	VAR jointtarget CDP_2918 := [[-11.73, 36.5, 4.79, 0, 48.7, -293.98], [9E9, 9E9, 9E9, 9E9, 9E9, 9E9]];
	VAR jointtarget CDP_2919 := [[-11.74, 36.51, 4.78, 0, 48.71, -294.65], [9E9, 9E9, 9E9, 9E9, 9E9, 9E9]];
	VAR jointtarget CDP_2920 := [[-11.8, 36.54, 4.72, 0, 48.73, -295.04], [9E9, 9E9, 9E9, 9E9, 9E9, 9E9]];
	VAR jointtarget CDP_2921 := [[-11.86, 36.57, 4.67, 0, 48.76, -295.11], [9E9, 9E9, 9E9, 9E9, 9E9, 9E9]];
	VAR jointtarget CDP_2922 := [[-11.93, 36.61, 4.62, 0, 48.78, -295.17], [9E9, 9E9, 9E9, 9E9, 9E9, 9E9]];
	VAR jointtarget CDP_2923 := [[-11.99, 36.64, 4.56, 0, 48.8, -295.23], [9E9, 9E9, 9E9, 9E9, 9E9, 9E9]];
	VAR jointtarget CDP_2924 := [[-12.05, 36.67, 4.51, 0, 48.82, -295.29], [9E9, 9E9, 9E9, 9E9, 9E9, 9E9]];
	VAR jointtarget CDP_2925 := [[-12.11, 36.7, 4.45, 0, 48.85, -295.35], [9E9, 9E9, 9E9, 9E9, 9E9, 9E9]];
	VAR jointtarget CDP_2926 := [[-12.17, 36.73, 4.4, 0, 48.87, -295.41], [9E9, 9E9, 9E9, 9E9, 9E9, 9E9]];
	VAR jointtarget CDP_2927 := [[-12.23, 36.76, 4.35, 0, 48.89, -295.47], [9E9, 9E9, 9E9, 9E9, 9E9, 9E9]];
	VAR jointtarget CDP_2928 := [[-12.29, 36.8, 4.29, 0, 48.91, -295.53], [9E9, 9E9, 9E9, 9E9, 9E9, 9E9]];
	VAR jointtarget CDP_2929 := [[-12.35, 36.83, 4.24, 0, 48.94, -295.59], [9E9, 9E9, 9E9, 9E9, 9E9, 9E9]];
	VAR jointtarget CDP_2930 := [[-12.41, 36.86, 4.18, 0, 48.96, -295.65], [9E9, 9E9, 9E9, 9E9, 9E9, 9E9]];
	VAR jointtarget CDP_2931 := [[-12.47, 36.89, 4.13, 0, 48.98, -295.71], [9E9, 9E9, 9E9, 9E9, 9E9, 9E9]];
	VAR jointtarget CDP_2932 := [[-12.53, 36.92, 4.07, 0, 49.01, -295.77], [9E9, 9E9, 9E9, 9E9, 9E9, 9E9]];
	VAR jointtarget CDP_2933 := [[-12.59, 36.96, 4.01, 0, 49.03, -295.83], [9E9, 9E9, 9E9, 9E9, 9E9, 9E9]];
	VAR jointtarget CDP_2934 := [[-12.65, 36.99, 3.96, 0, 49.05, -295.89], [9E9, 9E9, 9E9, 9E9, 9E9, 9E9]];
	VAR jointtarget CDP_2935 := [[-12.71, 37.02, 3.9, 0, 49.08, -295.95], [9E9, 9E9, 9E9, 9E9, 9E9, 9E9]];
	VAR jointtarget CDP_2936 := [[-12.77, 37.05, 3.85, 0, 49.1, -296.01], [9E9, 9E9, 9E9, 9E9, 9E9, 9E9]];
	VAR jointtarget CDP_2937 := [[-12.83, 37.09, 3.79, 0, 49.12, -296.07], [9E9, 9E9, 9E9, 9E9, 9E9, 9E9]];
	VAR jointtarget CDP_2938 := [[-12.89, 37.12, 3.73, 0, 49.15, -296.13], [9E9, 9E9, 9E9, 9E9, 9E9, 9E9]];
	VAR jointtarget CDP_2939 := [[-12.95, 37.15, 3.68, 0, 49.17, -296.19], [9E9, 9E9, 9E9, 9E9, 9E9, 9E9]];
	VAR jointtarget CDP_2940 := [[-13.07, 37.2, 3.59, 0, 49.21, -291.14], [9E9, 9E9, 9E9, 9E9, 9E9, 9E9]];
	VAR jointtarget CDP_2941 := [[-13.19, 37.23, 3.54, 0, 49.23, -280.95], [9E9, 9E9, 9E9, 9E9, 9E9, 9E9]];
	VAR jointtarget CDP_2942 := [[-13.32, 37.23, 3.54, 0, 49.23, -270.75], [9E9, 9E9, 9E9, 9E9, 9E9, 9E9]];
	VAR jointtarget CDP_2943 := [[-13.45, 37.21, 3.58, 0, 49.21, -260.55], [9E9, 9E9, 9E9, 9E9, 9E9, 9E9]];
	VAR jointtarget CDP_2944 := [[-13.57, 37.16, 3.66, 0, 49.18, -250.35], [9E9, 9E9, 9E9, 9E9, 9E9, 9E9]];
	VAR jointtarget CDP_2945 := [[-13.68, 37.09, 3.79, 0, 49.13, -240.14], [9E9, 9E9, 9E9, 9E9, 9E9, 9E9]];
	VAR jointtarget CDP_2946 := [[-13.78, 36.99, 3.95, 0, 49.06, -229.91], [9E9, 9E9, 9E9, 9E9, 9E9, 9E9]];
	VAR jointtarget CDP_2947 := [[-13.86, 36.88, 4.14, 0, 48.98, -219.67], [9E9, 9E9, 9E9, 9E9, 9E9, 9E9]];
	VAR jointtarget CDP_2948 := [[-13.93, 36.76, 4.35, 0, 48.89, -209.41], [9E9, 9E9, 9E9, 9E9, 9E9, 9E9]];
	VAR jointtarget CDP_2949 := [[-13.97, 36.62, 4.59, 0, 48.79, -199.13], [9E9, 9E9, 9E9, 9E9, 9E9, 9E9]];
	VAR jointtarget CDP_2950 := [[-13.99, 36.48, 4.83, 0, 48.69, -188.83], [9E9, 9E9, 9E9, 9E9, 9E9, 9E9]];
	VAR jointtarget CDP_2951 := [[-13.98, 36.34, 5.08, 0, 48.59, -178.5], [9E9, 9E9, 9E9, 9E9, 9E9, 9E9]];
	VAR jointtarget CDP_2952 := [[-13.96, 36.2, 5.32, 0, 48.48, -168.15], [9E9, 9E9, 9E9, 9E9, 9E9, 9E9]];
	VAR jointtarget CDP_2953 := [[-13.91, 36.06, 5.54, 0, 48.39, -157.77], [9E9, 9E9, 9E9, 9E9, 9E9, 9E9]];
	VAR jointtarget CDP_2954 := [[-13.84, 35.94, 5.75, 0, 48.3, -147.38], [9E9, 9E9, 9E9, 9E9, 9E9, 9E9]];
	VAR jointtarget CDP_2955 := [[-13.75, 35.84, 5.93, 0, 48.23, -136.97], [9E9, 9E9, 9E9, 9E9, 9E9, 9E9]];
	VAR jointtarget CDP_2956 := [[-13.64, 35.75, 6.08, 0, 48.17, -126.54], [9E9, 9E9, 9E9, 9E9, 9E9, 9E9]];
	VAR jointtarget CDP_2957 := [[-13.52, 35.69, 6.18, 0, 48.13, -116.09], [9E9, 9E9, 9E9, 9E9, 9E9, 9E9]];
	VAR jointtarget CDP_2958 := [[-13.4, 35.65, 6.25, 0, 48.1, -105.64], [9E9, 9E9, 9E9, 9E9, 9E9, 9E9]];
	VAR jointtarget CDP_2959 := [[-13.27, 35.64, 6.27, 0, 48.09, -95.19], [9E9, 9E9, 9E9, 9E9, 9E9, 9E9]];
	VAR jointtarget CDP_2960 := [[-13.2, 35.64, 6.27, 0, 48.09, -89.96], [9E9, 9E9, 9E9, 9E9, 9E9, 9E9]];
	VAR jointtarget CDP_2961 := [[-13.13, 35.64, 6.27, 0, 48.09, -89.89], [9E9, 9E9, 9E9, 9E9, 9E9, 9E9]];
	VAR jointtarget CDP_2962 := [[-13.06, 35.64, 6.27, 0, 48.09, -89.82], [9E9, 9E9, 9E9, 9E9, 9E9, 9E9]];
	VAR jointtarget CDP_2963 := [[-12.99, 35.64, 6.27, 0, 48.09, -89.75], [9E9, 9E9, 9E9, 9E9, 9E9, 9E9]];
	VAR jointtarget CDP_2964 := [[-12.93, 35.64, 6.27, 0, 48.09, -89.69], [9E9, 9E9, 9E9, 9E9, 9E9, 9E9]];
	VAR jointtarget CDP_2965 := [[-12.86, 35.64, 6.27, 0, 48.09, -89.62], [9E9, 9E9, 9E9, 9E9, 9E9, 9E9]];
	VAR jointtarget CDP_2966 := [[-12.79, 35.64, 6.27, 0, 48.09, -89.55], [9E9, 9E9, 9E9, 9E9, 9E9, 9E9]];
	VAR jointtarget CDP_2967 := [[-12.72, 35.64, 6.27, 0, 48.1, -89.48], [9E9, 9E9, 9E9, 9E9, 9E9, 9E9]];
	VAR jointtarget CDP_2968 := [[-12.65, 35.64, 6.26, 0, 48.1, -89.41], [9E9, 9E9, 9E9, 9E9, 9E9, 9E9]];
	VAR jointtarget CDP_2969 := [[-12.59, 35.64, 6.26, 0, 48.1, -89.35], [9E9, 9E9, 9E9, 9E9, 9E9, 9E9]];
	VAR jointtarget CDP_2970 := [[-12.52, 35.64, 6.26, 0, 48.1, -89.28], [9E9, 9E9, 9E9, 9E9, 9E9, 9E9]];
	VAR jointtarget CDP_2971 := [[-12.45, 35.64, 6.26, 0, 48.1, -89.21], [9E9, 9E9, 9E9, 9E9, 9E9, 9E9]];
	VAR jointtarget CDP_2972 := [[-12.38, 35.64, 6.26, 0, 48.1, -89.14], [9E9, 9E9, 9E9, 9E9, 9E9, 9E9]];
	VAR jointtarget CDP_2973 := [[-12.32, 35.64, 6.26, 0, 48.1, -89.07], [9E9, 9E9, 9E9, 9E9, 9E9, 9E9]];
	VAR jointtarget CDP_2974 := [[-12.25, 35.64, 6.25, 0, 48.11, -89.01], [9E9, 9E9, 9E9, 9E9, 9E9, 9E9]];
	VAR jointtarget CDP_2975 := [[-12.18, 35.64, 6.25, 0, 48.11, -88.94], [9E9, 9E9, 9E9, 9E9, 9E9, 9E9]];
	VAR jointtarget CDP_2976 := [[-12.11, 35.64, 6.25, 0, 48.11, -88.87], [9E9, 9E9, 9E9, 9E9, 9E9, 9E9]];
	VAR jointtarget CDP_2977 := [[-12.04, 35.64, 6.25, 0, 48.11, -88.8], [9E9, 9E9, 9E9, 9E9, 9E9, 9E9]];
	VAR jointtarget CDP_2978 := [[-11.98, 35.64, 6.24, 0, 48.11, -88.74], [9E9, 9E9, 9E9, 9E9, 9E9, 9E9]];
	VAR jointtarget CDP_2979 := [[-11.91, 35.65, 6.24, 0, 48.11, -88.67], [9E9, 9E9, 9E9, 9E9, 9E9, 9E9]];
	VAR jointtarget CDP_2980 := [[-11.89, 35.65, 6.24, 0, 48.11, -88.98], [9E9, 9E9, 9E9, 9E9, 9E9, 9E9]];
	VAR jointtarget CDP_2981 := [[-11.87, 35.65, 6.24, 0, 48.11, -89.63], [9E9, 9E9, 9E9, 9E9, 9E9, 9E9]];
	VAR jointtarget CDP_2982 := [[-11.86, 35.65, 6.24, 0, 48.11, -90.27], [9E9, 9E9, 9E9, 9E9, 9E9, 9E9]];
	VAR jointtarget CDP_2983 := [[-11.84, 35.65, 6.24, 0, 48.11, -90.92], [9E9, 9E9, 9E9, 9E9, 9E9, 9E9]];
	VAR jointtarget CDP_2984 := [[-11.82, 35.64, 6.24, 0, 48.11, -91.56], [9E9, 9E9, 9E9, 9E9, 9E9, 9E9]];
	VAR jointtarget CDP_2985 := [[-11.81, 35.64, 6.24, 0, 48.11, -92.21], [9E9, 9E9, 9E9, 9E9, 9E9, 9E9]];
	VAR jointtarget CDP_2986 := [[-11.79, 35.64, 6.24, 0, 48.11, -92.85], [9E9, 9E9, 9E9, 9E9, 9E9, 9E9]];
	VAR jointtarget CDP_2987 := [[-11.77, 35.64, 6.25, 0, 48.11, -93.5], [9E9, 9E9, 9E9, 9E9, 9E9, 9E9]];
	VAR jointtarget CDP_2988 := [[-11.76, 35.64, 6.25, 0, 48.11, -94.14], [9E9, 9E9, 9E9, 9E9, 9E9, 9E9]];
	VAR jointtarget CDP_2989 := [[-11.74, 35.64, 6.25, 0, 48.11, -94.79], [9E9, 9E9, 9E9, 9E9, 9E9, 9E9]];
	VAR jointtarget CDP_2990 := [[-11.72, 35.64, 6.25, 0, 48.11, -95.43], [9E9, 9E9, 9E9, 9E9, 9E9, 9E9]];
	VAR jointtarget CDP_2991 := [[-11.71, 35.63, 6.26, 0, 48.11, -96.08], [9E9, 9E9, 9E9, 9E9, 9E9, 9E9]];
	VAR jointtarget CDP_2992 := [[-11.69, 35.63, 6.26, 0, 48.11, -96.72], [9E9, 9E9, 9E9, 9E9, 9E9, 9E9]];
	VAR jointtarget CDP_2993 := [[-11.67, 35.63, 6.26, 0, 48.11, -97.37], [9E9, 9E9, 9E9, 9E9, 9E9, 9E9]];
	VAR jointtarget CDP_2994 := [[-11.66, 35.63, 6.27, 0, 48.1, -98.01], [9E9, 9E9, 9E9, 9E9, 9E9, 9E9]];
	VAR jointtarget CDP_2995 := [[-11.64, 35.62, 6.27, 0, 48.1, -98.66], [9E9, 9E9, 9E9, 9E9, 9E9, 9E9]];
	VAR jointtarget CDP_2996 := [[-11.62, 35.62, 6.28, 0, 48.1, -99.31], [9E9, 9E9, 9E9, 9E9, 9E9, 9E9]];
	VAR jointtarget CDP_2997 := [[-11.61, 35.62, 6.28, 0, 48.1, -99.95], [9E9, 9E9, 9E9, 9E9, 9E9, 9E9]];
	VAR jointtarget CDP_2998 := [[-11.59, 35.62, 6.29, 0, 48.1, -100.6], [9E9, 9E9, 9E9, 9E9, 9E9, 9E9]];
	VAR jointtarget CDP_2999 := [[-11.57, 35.61, 6.3, 0, 48.09, -101.24], [9E9, 9E9, 9E9, 9E9, 9E9, 9E9]];
	VAR jointtarget CDP_3000 := [[-10.48, 35.38, 6.69, 0, 47.93, -100.48], [9E9, 9E9, 9E9, 9E9, 9E9, 9E9]];
	VAR jointtarget CDP_3001 := [[-9.38, 35.18, 7.04, 0, 47.78, -99.38], [9E9, 9E9, 9E9, 9E9, 9E9, 9E9]];
	VAR jointtarget CDP_3002 := [[-8.27, 34.99, 7.35, 0, 47.66, -98.27], [9E9, 9E9, 9E9, 9E9, 9E9, 9E9]];
	VAR jointtarget CDP_3003 := [[-7.15, 34.83, 7.62, 0, 47.54, -97.15], [9E9, 9E9, 9E9, 9E9, 9E9, 9E9]];
	VAR jointtarget CDP_3004 := [[-6.03, 34.7, 7.86, 0, 47.45, -96.03], [9E9, 9E9, 9E9, 9E9, 9E9, 9E9]];
	VAR jointtarget CDP_3005 := [[-4.9, 34.58, 8.05, 0, 47.37, -94.9], [9E9, 9E9, 9E9, 9E9, 9E9, 9E9]];
	VAR jointtarget CDP_3006 := [[-3.77, 34.49, 8.2, 0, 47.31, -93.77], [9E9, 9E9, 9E9, 9E9, 9E9, 9E9]];
	VAR jointtarget CDP_3007 := [[-2.64, 34.43, 8.32, 0, 47.26, -92.64], [9E9, 9E9, 9E9, 9E9, 9E9, 9E9]];
	VAR jointtarget CDP_3008 := [[-1.51, 34.38, 8.39, 0, 47.23, -91.51], [9E9, 9E9, 9E9, 9E9, 9E9, 9E9]];
	VAR jointtarget CDP_3009 := [[-0.37, 34.36, 8.42, 0, 47.22, -90.37], [9E9, 9E9, 9E9, 9E9, 9E9, 9E9]];
	VAR jointtarget CDP_3010 := [[0.76, 34.37, 8.41, 0, 47.22, -89.24], [9E9, 9E9, 9E9, 9E9, 9E9, 9E9]];
	VAR jointtarget CDP_3011 := [[1.9, 34.39, 8.37, 0, 47.24, -88.1], [9E9, 9E9, 9E9, 9E9, 9E9, 9E9]];
	VAR jointtarget CDP_3012 := [[3.03, 34.45, 8.28, 0, 47.27, -86.97], [9E9, 9E9, 9E9, 9E9, 9E9, 9E9]];
	VAR jointtarget CDP_3013 := [[4.16, 34.52, 8.15, 0, 47.33, -85.84], [9E9, 9E9, 9E9, 9E9, 9E9, 9E9]];
	VAR jointtarget CDP_3014 := [[5.29, 34.62, 7.99, 0, 47.39, -84.71], [9E9, 9E9, 9E9, 9E9, 9E9, 9E9]];
	VAR jointtarget CDP_3015 := [[6.42, 34.74, 7.78, 0, 47.48, -83.58], [9E9, 9E9, 9E9, 9E9, 9E9, 9E9]];
	VAR jointtarget CDP_3016 := [[7.54, 34.89, 7.53, 0, 47.58, -82.46], [9E9, 9E9, 9E9, 9E9, 9E9, 9E9]];
	VAR jointtarget CDP_3017 := [[8.65, 35.05, 7.25, 0, 47.7, -81.35], [9E9, 9E9, 9E9, 9E9, 9E9, 9E9]];
	VAR jointtarget CDP_3018 := [[9.76, 35.24, 6.92, 0, 47.83, -80.24], [9E9, 9E9, 9E9, 9E9, 9E9, 9E9]];
	VAR jointtarget CDP_3019 := [[10.86, 35.46, 6.56, 0, 47.98, -79.14], [9E9, 9E9, 9E9, 9E9, 9E9, 9E9]];
	VAR jointtarget CDP_3020 := [[10.87, 35.46, 6.55, 0, 47.99, -79.46], [9E9, 9E9, 9E9, 9E9, 9E9, 9E9]];
	VAR jointtarget CDP_3021 := [[10.89, 35.47, 6.55, 0, 47.99, -80.1], [9E9, 9E9, 9E9, 9E9, 9E9, 9E9]];
	VAR jointtarget CDP_3022 := [[10.91, 35.47, 6.54, 0, 47.99, -80.75], [9E9, 9E9, 9E9, 9E9, 9E9, 9E9]];
	VAR jointtarget CDP_3023 := [[10.92, 35.47, 6.54, 0, 47.99, -81.39], [9E9, 9E9, 9E9, 9E9, 9E9, 9E9]];
	VAR jointtarget CDP_3024 := [[10.94, 35.47, 6.53, 0, 48, -82.04], [9E9, 9E9, 9E9, 9E9, 9E9, 9E9]];
	VAR jointtarget CDP_3025 := [[10.96, 35.48, 6.53, 0, 48, -82.68], [9E9, 9E9, 9E9, 9E9, 9E9, 9E9]];
	VAR jointtarget CDP_3026 := [[10.97, 35.48, 6.52, 0, 48, -83.33], [9E9, 9E9, 9E9, 9E9, 9E9, 9E9]];
	VAR jointtarget CDP_3027 := [[10.99, 35.48, 6.52, 0, 48, -83.97], [9E9, 9E9, 9E9, 9E9, 9E9, 9E9]];
	VAR jointtarget CDP_3028 := [[11.01, 35.48, 6.52, 0, 48, -84.62], [9E9, 9E9, 9E9, 9E9, 9E9, 9E9]];
	VAR jointtarget CDP_3029 := [[11.02, 35.48, 6.52, 0, 48, -85.27], [9E9, 9E9, 9E9, 9E9, 9E9, 9E9]];
	VAR jointtarget CDP_3030 := [[11.04, 35.48, 6.51, 0, 48, -85.91], [9E9, 9E9, 9E9, 9E9, 9E9, 9E9]];
	VAR jointtarget CDP_3031 := [[11.06, 35.49, 6.51, 0, 48, -86.56], [9E9, 9E9, 9E9, 9E9, 9E9, 9E9]];
	VAR jointtarget CDP_3032 := [[11.07, 35.49, 6.51, 0, 48, -87.2], [9E9, 9E9, 9E9, 9E9, 9E9, 9E9]];
	VAR jointtarget CDP_3033 := [[11.09, 35.49, 6.51, 0, 48, -87.85], [9E9, 9E9, 9E9, 9E9, 9E9, 9E9]];
	VAR jointtarget CDP_3034 := [[11.11, 35.49, 6.51, 0, 48, -88.49], [9E9, 9E9, 9E9, 9E9, 9E9, 9E9]];
	VAR jointtarget CDP_3035 := [[11.13, 35.49, 6.51, 0, 48.01, -89.14], [9E9, 9E9, 9E9, 9E9, 9E9, 9E9]];
	VAR jointtarget CDP_3036 := [[11.14, 35.49, 6.51, 0, 48.01, -89.78], [9E9, 9E9, 9E9, 9E9, 9E9, 9E9]];
	VAR jointtarget CDP_3037 := [[11.16, 35.49, 6.51, 0, 48.01, -90.43], [9E9, 9E9, 9E9, 9E9, 9E9, 9E9]];
	VAR jointtarget CDP_3038 := [[11.18, 35.49, 6.51, 0, 48, -91.07], [9E9, 9E9, 9E9, 9E9, 9E9, 9E9]];
	VAR jointtarget CDP_3039 := [[11.19, 35.49, 6.51, 0, 48, -91.72], [9E9, 9E9, 9E9, 9E9, 9E9, 9E9]];
	VAR jointtarget CDP_3040 := [[11.26, 35.48, 6.51, 0, 48, -91.98], [9E9, 9E9, 9E9, 9E9, 9E9, 9E9]];
	VAR jointtarget CDP_3041 := [[11.33, 35.48, 6.52, 0, 48, -91.91], [9E9, 9E9, 9E9, 9E9, 9E9, 9E9]];
	VAR jointtarget CDP_3042 := [[11.4, 35.48, 6.52, 0, 48, -91.84], [9E9, 9E9, 9E9, 9E9, 9E9, 9E9]];
	VAR jointtarget CDP_3043 := [[11.47, 35.48, 6.53, 0, 48, -91.78], [9E9, 9E9, 9E9, 9E9, 9E9, 9E9]];
	VAR jointtarget CDP_3044 := [[11.53, 35.47, 6.53, 0, 48, -91.71], [9E9, 9E9, 9E9, 9E9, 9E9, 9E9]];
	VAR jointtarget CDP_3045 := [[11.6, 35.47, 6.53, 0, 47.99, -91.64], [9E9, 9E9, 9E9, 9E9, 9E9, 9E9]];
	VAR jointtarget CDP_3046 := [[11.67, 35.47, 6.54, 0, 47.99, -91.57], [9E9, 9E9, 9E9, 9E9, 9E9, 9E9]];
	VAR jointtarget CDP_3047 := [[11.74, 35.47, 6.54, 0, 47.99, -91.5], [9E9, 9E9, 9E9, 9E9, 9E9, 9E9]];
	VAR jointtarget CDP_3048 := [[11.81, 35.47, 6.54, 0, 47.99, -91.44], [9E9, 9E9, 9E9, 9E9, 9E9, 9E9]];
	VAR jointtarget CDP_3049 := [[11.87, 35.46, 6.55, 0, 47.99, -91.37], [9E9, 9E9, 9E9, 9E9, 9E9, 9E9]];
	VAR jointtarget CDP_3050 := [[11.94, 35.46, 6.55, 0, 47.99, -91.3], [9E9, 9E9, 9E9, 9E9, 9E9, 9E9]];
	VAR jointtarget CDP_3051 := [[12.01, 35.46, 6.55, 0, 47.99, -91.23], [9E9, 9E9, 9E9, 9E9, 9E9, 9E9]];
	VAR jointtarget CDP_3052 := [[12.08, 35.46, 6.55, 0, 47.99, -91.16], [9E9, 9E9, 9E9, 9E9, 9E9, 9E9]];
	VAR jointtarget CDP_3053 := [[12.15, 35.46, 6.56, 0, 47.98, -91.09], [9E9, 9E9, 9E9, 9E9, 9E9, 9E9]];
	VAR jointtarget CDP_3054 := [[12.21, 35.46, 6.56, 0, 47.98, -91.03], [9E9, 9E9, 9E9, 9E9, 9E9, 9E9]];
	VAR jointtarget CDP_3055 := [[12.28, 35.46, 6.56, 0, 47.98, -90.96], [9E9, 9E9, 9E9, 9E9, 9E9, 9E9]];
	VAR jointtarget CDP_3056 := [[12.35, 35.45, 6.56, 0, 47.98, -90.89], [9E9, 9E9, 9E9, 9E9, 9E9, 9E9]];
	VAR jointtarget CDP_3057 := [[12.42, 35.45, 6.57, 0, 47.98, -90.82], [9E9, 9E9, 9E9, 9E9, 9E9, 9E9]];
	VAR jointtarget CDP_3058 := [[12.49, 35.45, 6.57, 0, 47.98, -90.75], [9E9, 9E9, 9E9, 9E9, 9E9, 9E9]];
	VAR jointtarget CDP_3059 := [[12.55, 35.45, 6.57, 0, 47.98, -90.69], [9E9, 9E9, 9E9, 9E9, 9E9, 9E9]];
	VAR jointtarget CDP_3060 := [[12.69, 35.46, 6.55, 0, 47.99, -85.39], [9E9, 9E9, 9E9, 9E9, 9E9, 9E9]];
	VAR jointtarget CDP_3061 := [[12.81, 35.5, 6.49, 0, 48.01, -74.94], [9E9, 9E9, 9E9, 9E9, 9E9, 9E9]];
	VAR jointtarget CDP_3062 := [[12.93, 35.56, 6.38, 0, 48.06, -64.5], [9E9, 9E9, 9E9, 9E9, 9E9, 9E9]];
	VAR jointtarget CDP_3063 := [[13.04, 35.64, 6.24, 0, 48.12, -54.07], [9E9, 9E9, 9E9, 9E9, 9E9, 9E9]];
	VAR jointtarget CDP_3064 := [[13.13, 35.75, 6.06, 0, 48.19, -43.65], [9E9, 9E9, 9E9, 9E9, 9E9, 9E9]];
	VAR jointtarget CDP_3065 := [[13.2, 35.87, 5.86, 0, 48.27, -33.25], [9E9, 9E9, 9E9, 9E9, 9E9, 9E9]];
	VAR jointtarget CDP_3066 := [[13.25, 36, 5.63, 0, 48.37, -22.88], [9E9, 9E9, 9E9, 9E9, 9E9, 9E9]];
	VAR jointtarget CDP_3067 := [[13.28, 36.14, 5.39, 0, 48.47, -12.53], [9E9, 9E9, 9E9, 9E9, 9E9, 9E9]];
	VAR jointtarget CDP_3068 := [[13.29, 36.28, 5.15, 0, 48.57, -2.2], [9E9, 9E9, 9E9, 9E9, 9E9, 9E9]];
	VAR jointtarget CDP_3069 := [[13.27, 36.42, 4.91, 0, 48.67, 8.11], [9E9, 9E9, 9E9, 9E9, 9E9, 9E9]];
	VAR jointtarget CDP_3070 := [[13.23, 36.56, 4.67, 0, 48.77, 18.39], [9E9, 9E9, 9E9, 9E9, 9E9, 9E9]];
	VAR jointtarget CDP_3071 := [[13.17, 36.68, 4.46, 0, 48.86, 28.65], [9E9, 9E9, 9E9, 9E9, 9E9, 9E9]];
	VAR jointtarget CDP_3072 := [[13.08, 36.8, 4.26, 0, 48.94, 38.9], [9E9, 9E9, 9E9, 9E9, 9E9, 9E9]];
	VAR jointtarget CDP_3073 := [[12.99, 36.89, 4.1, 0, 49.01, 49.12], [9E9, 9E9, 9E9, 9E9, 9E9, 9E9]];
	VAR jointtarget CDP_3074 := [[12.88, 36.96, 3.98, 0, 49.06, 59.33], [9E9, 9E9, 9E9, 9E9, 9E9, 9E9]];
	VAR jointtarget CDP_3075 := [[12.75, 37.01, 3.89, 0, 49.1, 69.54], [9E9, 9E9, 9E9, 9E9, 9E9, 9E9]];
	VAR jointtarget CDP_3076 := [[12.63, 37.04, 3.84, 0, 49.12, 79.73], [9E9, 9E9, 9E9, 9E9, 9E9, 9E9]];
	VAR jointtarget CDP_3077 := [[12.5, 37.04, 3.84, 0, 49.12, 89.93], [9E9, 9E9, 9E9, 9E9, 9E9, 9E9]];
	VAR jointtarget CDP_3078 := [[12.37, 37.01, 3.89, 0, 49.1, 100.13], [9E9, 9E9, 9E9, 9E9, 9E9, 9E9]];
	VAR jointtarget CDP_3079 := [[12.25, 36.96, 3.97, 0, 49.06, 110.33], [9E9, 9E9, 9E9, 9E9, 9E9, 9E9]];
	VAR jointtarget CDP_3080 := [[12.19, 36.93, 4.03, 0, 49.04, 115.43], [9E9, 9E9, 9E9, 9E9, 9E9, 9E9]];
	VAR jointtarget CDP_3081 := [[12.13, 36.9, 4.08, 0, 49.01, 115.37], [9E9, 9E9, 9E9, 9E9, 9E9, 9E9]];
	VAR jointtarget CDP_3082 := [[12.07, 36.87, 4.14, 0, 48.99, 115.31], [9E9, 9E9, 9E9, 9E9, 9E9, 9E9]];
	VAR jointtarget CDP_3083 := [[12.01, 36.84, 4.19, 0, 48.97, 115.25], [9E9, 9E9, 9E9, 9E9, 9E9, 9E9]];
	VAR jointtarget CDP_3084 := [[11.95, 36.81, 4.25, 0, 48.95, 115.19], [9E9, 9E9, 9E9, 9E9, 9E9, 9E9]];
	VAR jointtarget CDP_3085 := [[11.89, 36.77, 4.3, 0, 48.92, 115.13], [9E9, 9E9, 9E9, 9E9, 9E9, 9E9]];
	VAR jointtarget CDP_3086 := [[11.83, 36.74, 4.36, 0, 48.9, 115.07], [9E9, 9E9, 9E9, 9E9, 9E9, 9E9]];
	VAR jointtarget CDP_3087 := [[11.77, 36.71, 4.41, 0, 48.88, 115.01], [9E9, 9E9, 9E9, 9E9, 9E9, 9E9]];
	VAR jointtarget CDP_3088 := [[11.71, 36.68, 4.46, 0, 48.86, 114.95], [9E9, 9E9, 9E9, 9E9, 9E9, 9E9]];
	VAR jointtarget CDP_3089 := [[11.65, 36.65, 4.52, 0, 48.83, 114.89], [9E9, 9E9, 9E9, 9E9, 9E9, 9E9]];
	VAR jointtarget CDP_3090 := [[11.59, 36.62, 4.57, 0, 48.81, 114.83], [9E9, 9E9, 9E9, 9E9, 9E9, 9E9]];
	VAR jointtarget CDP_3091 := [[11.53, 36.59, 4.62, 0, 48.79, 114.77], [9E9, 9E9, 9E9, 9E9, 9E9, 9E9]];
	VAR jointtarget CDP_3092 := [[11.47, 36.56, 4.68, 0, 48.77, 114.71], [9E9, 9E9, 9E9, 9E9, 9E9, 9E9]];
	VAR jointtarget CDP_3093 := [[11.4, 36.53, 4.73, 0, 48.74, 114.64], [9E9, 9E9, 9E9, 9E9, 9E9, 9E9]];
	VAR jointtarget CDP_3094 := [[11.34, 36.49, 4.78, 0, 48.72, 114.58], [9E9, 9E9, 9E9, 9E9, 9E9, 9E9]];
	VAR jointtarget CDP_3095 := [[11.28, 36.46, 4.83, 0, 48.7, 114.52], [9E9, 9E9, 9E9, 9E9, 9E9, 9E9]];
	VAR jointtarget CDP_3096 := [[11.22, 36.43, 4.89, 0, 48.68, 114.46], [9E9, 9E9, 9E9, 9E9, 9E9, 9E9]];
	VAR jointtarget CDP_3097 := [[11.16, 36.4, 4.94, 0, 48.66, 114.4], [9E9, 9E9, 9E9, 9E9, 9E9, 9E9]];
	VAR jointtarget CDP_3098 := [[11.1, 36.37, 4.99, 0, 48.64, 114.34], [9E9, 9E9, 9E9, 9E9, 9E9, 9E9]];
	VAR jointtarget CDP_3099 := [[11.04, 36.34, 5.04, 0, 48.61, 114.28], [9E9, 9E9, 9E9, 9E9, 9E9, 9E9]];
	VAR jointtarget CDP_3100 := [[11.02, 36.33, 5.06, 0, 48.61, 113.93], [9E9, 9E9, 9E9, 9E9, 9E9, 9E9]];
	VAR jointtarget CDP_3101 := [[11.01, 36.33, 5.07, 0, 48.6, 113.26], [9E9, 9E9, 9E9, 9E9, 9E9, 9E9]];
	VAR jointtarget CDP_3102 := [[10.99, 36.32, 5.08, 0, 48.6, 112.58], [9E9, 9E9, 9E9, 9E9, 9E9, 9E9]];
	VAR jointtarget CDP_3103 := [[10.98, 36.31, 5.09, 0, 48.59, 111.9], [9E9, 9E9, 9E9, 9E9, 9E9, 9E9]];
	VAR jointtarget CDP_3104 := [[10.96, 36.31, 5.1, 0, 48.59, 111.22], [9E9, 9E9, 9E9, 9E9, 9E9, 9E9]];
	VAR jointtarget CDP_3105 := [[10.95, 36.3, 5.12, 0, 48.58, 110.55], [9E9, 9E9, 9E9, 9E9, 9E9, 9E9]];
	VAR jointtarget CDP_3106 := [[10.93, 36.29, 5.13, 0, 48.58, 109.87], [9E9, 9E9, 9E9, 9E9, 9E9, 9E9]];
	VAR jointtarget CDP_3107 := [[10.91, 36.29, 5.14, 0, 48.58, 109.19], [9E9, 9E9, 9E9, 9E9, 9E9, 9E9]];
	VAR jointtarget CDP_3108 := [[10.9, 36.28, 5.15, 0, 48.57, 108.51], [9E9, 9E9, 9E9, 9E9, 9E9, 9E9]];
	VAR jointtarget CDP_3109 := [[10.88, 36.28, 5.16, 0, 48.57, 107.83], [9E9, 9E9, 9E9, 9E9, 9E9, 9E9]];
	VAR jointtarget CDP_3110 := [[10.87, 36.27, 5.17, 0, 48.56, 107.16], [9E9, 9E9, 9E9, 9E9, 9E9, 9E9]];
	VAR jointtarget CDP_3111 := [[10.85, 36.27, 5.17, 0, 48.56, 106.48], [9E9, 9E9, 9E9, 9E9, 9E9, 9E9]];
	VAR jointtarget CDP_3112 := [[10.83, 36.26, 5.18, 0, 48.56, 105.8], [9E9, 9E9, 9E9, 9E9, 9E9, 9E9]];
	VAR jointtarget CDP_3113 := [[10.82, 36.26, 5.19, 0, 48.55, 105.12], [9E9, 9E9, 9E9, 9E9, 9E9, 9E9]];
	VAR jointtarget CDP_3114 := [[10.8, 36.25, 5.2, 0, 48.55, 104.44], [9E9, 9E9, 9E9, 9E9, 9E9, 9E9]];
	VAR jointtarget CDP_3115 := [[10.79, 36.25, 5.21, 0, 48.55, 103.77], [9E9, 9E9, 9E9, 9E9, 9E9, 9E9]];
	VAR jointtarget CDP_3116 := [[10.77, 36.24, 5.21, 0, 48.54, 103.09], [9E9, 9E9, 9E9, 9E9, 9E9, 9E9]];
	VAR jointtarget CDP_3117 := [[10.75, 36.24, 5.22, 0, 48.54, 102.41], [9E9, 9E9, 9E9, 9E9, 9E9, 9E9]];
	VAR jointtarget CDP_3118 := [[10.74, 36.24, 5.23, 0, 48.54, 101.73], [9E9, 9E9, 9E9, 9E9, 9E9, 9E9]];
	VAR jointtarget CDP_3119 := [[10.72, 36.23, 5.23, 0, 48.54, 101.05], [9E9, 9E9, 9E9, 9E9, 9E9, 9E9]];
	VAR jointtarget CDP_3120 := [[9.64, 36.02, 5.59, 0, 48.38, 99.64], [9E9, 9E9, 9E9, 9E9, 9E9, 9E9]];
	VAR jointtarget CDP_3121 := [[8.56, 35.83, 5.92, 0, 48.25, 98.56], [9E9, 9E9, 9E9, 9E9, 9E9, 9E9]];
	VAR jointtarget CDP_3122 := [[7.47, 35.67, 6.2, 0, 48.13, 97.47], [9E9, 9E9, 9E9, 9E9, 9E9, 9E9]];
	VAR jointtarget CDP_3123 := [[6.38, 35.52, 6.45, 0, 48.03, 96.38], [9E9, 9E9, 9E9, 9E9, 9E9, 9E9]];
	VAR jointtarget CDP_3124 := [[5.28, 35.4, 6.65, 0, 47.95, 95.28], [9E9, 9E9, 9E9, 9E9, 9E9, 9E9]];
	VAR jointtarget CDP_3125 := [[4.17, 35.31, 6.82, 0, 47.88, 94.17], [9E9, 9E9, 9E9, 9E9, 9E9, 9E9]];
	VAR jointtarget CDP_3126 := [[3.07, 35.23, 6.95, 0, 47.82, 93.07], [9E9, 9E9, 9E9, 9E9, 9E9, 9E9]];
	VAR jointtarget CDP_3127 := [[1.96, 35.18, 7.04, 0, 47.79, 91.96], [9E9, 9E9, 9E9, 9E9, 9E9, 9E9]];
	VAR jointtarget CDP_3128 := [[0.85, 35.15, 7.08, 0, 47.77, 90.85], [9E9, 9E9, 9E9, 9E9, 9E9, 9E9]];
	VAR jointtarget CDP_3129 := [[-0.26, 35.14, 7.09, 0, 47.76, 89.74], [9E9, 9E9, 9E9, 9E9, 9E9, 9E9]];
	VAR jointtarget CDP_3130 := [[-1.37, 35.16, 7.07, 0, 47.77, 88.63], [9E9, 9E9, 9E9, 9E9, 9E9, 9E9]];
	VAR jointtarget CDP_3131 := [[-2.48, 35.2, 7, 0, 47.8, 87.52], [9E9, 9E9, 9E9, 9E9, 9E9, 9E9]];
	VAR jointtarget CDP_3132 := [[-3.59, 35.26, 6.89, 0, 47.85, 86.41], [9E9, 9E9, 9E9, 9E9, 9E9, 9E9]];
	VAR jointtarget CDP_3133 := [[-4.7, 35.35, 6.74, 0, 47.91, 85.3], [9E9, 9E9, 9E9, 9E9, 9E9, 9E9]];
	VAR jointtarget CDP_3134 := [[-5.8, 35.46, 6.56, 0, 47.98, 84.2], [9E9, 9E9, 9E9, 9E9, 9E9, 9E9]];
	VAR jointtarget CDP_3135 := [[-6.9, 35.59, 6.33, 0, 48.08, 83.1], [9E9, 9E9, 9E9, 9E9, 9E9, 9E9]];
	VAR jointtarget CDP_3136 := [[-7.99, 35.74, 6.07, 0, 48.19, 82.01], [9E9, 9E9, 9E9, 9E9, 9E9, 9E9]];
	VAR jointtarget CDP_3137 := [[-9.08, 35.92, 5.77, 0, 48.31, 80.92], [9E9, 9E9, 9E9, 9E9, 9E9, 9E9]];
	VAR jointtarget CDP_3138 := [[-10.16, 36.12, 5.43, 0, 48.45, 79.84], [9E9, 9E9, 9E9, 9E9, 9E9, 9E9]];
	VAR jointtarget CDP_3139 := [[-11.23, 36.34, 5.05, 0, 48.61, 78.77], [9E9, 9E9, 9E9, 9E9, 9E9, 9E9]];
	VAR jointtarget CDP_3140 := [[-11.28, 36.35, 5.03, 0, 48.62, 79.81], [9E9, 9E9, 9E9, 9E9, 9E9, 9E9]];
	VAR jointtarget CDP_3141 := [[-11.34, 36.36, 5.01, 0, 48.63, 81.95], [9E9, 9E9, 9E9, 9E9, 9E9, 9E9]];
	VAR jointtarget CDP_3142 := [[-11.39, 36.37, 5, 0, 48.63, 84.09], [9E9, 9E9, 9E9, 9E9, 9E9, 9E9]];
	VAR jointtarget CDP_3143 := [[-11.45, 36.37, 5, 0, 48.63, 86.23], [9E9, 9E9, 9E9, 9E9, 9E9, 9E9]];
	VAR jointtarget CDP_3144 := [[-11.5, 36.37, 4.99, 0, 48.63, 88.37], [9E9, 9E9, 9E9, 9E9, 9E9, 9E9]];
	VAR jointtarget CDP_3145 := [[-11.56, 36.37, 4.99, 0, 48.63, 90.51], [9E9, 9E9, 9E9, 9E9, 9E9, 9E9]];
	VAR jointtarget CDP_3146 := [[-11.61, 36.37, 5, 0, 48.63, 92.65], [9E9, 9E9, 9E9, 9E9, 9E9, 9E9]];
	VAR jointtarget CDP_3147 := [[-11.67, 36.36, 5.01, 0, 48.63, 94.78], [9E9, 9E9, 9E9, 9E9, 9E9, 9E9]];
	VAR jointtarget CDP_3148 := [[-11.72, 36.36, 5.02, 0, 48.62, 96.92], [9E9, 9E9, 9E9, 9E9, 9E9, 9E9]];
	VAR jointtarget CDP_3149 := [[-11.78, 36.35, 5.04, 0, 48.62, 99.06], [9E9, 9E9, 9E9, 9E9, 9E9, 9E9]];
	VAR jointtarget CDP_3150 := [[-11.83, 36.33, 5.06, 0, 48.61, 101.2], [9E9, 9E9, 9E9, 9E9, 9E9, 9E9]];
	VAR jointtarget CDP_3151 := [[-11.89, 36.32, 5.08, 0, 48.6, 103.34], [9E9, 9E9, 9E9, 9E9, 9E9, 9E9]];
	VAR jointtarget CDP_3152 := [[-11.94, 36.3, 5.11, 0, 48.59, 105.48], [9E9, 9E9, 9E9, 9E9, 9E9, 9E9]];
	VAR jointtarget CDP_3153 := [[-11.99, 36.29, 5.14, 0, 48.57, 107.63], [9E9, 9E9, 9E9, 9E9, 9E9, 9E9]];
	VAR jointtarget CDP_3154 := [[-12.04, 36.27, 5.18, 0, 48.56, 109.77], [9E9, 9E9, 9E9, 9E9, 9E9, 9E9]];
	VAR jointtarget CDP_3155 := [[-12.09, 36.24, 5.21, 0, 48.54, 111.91], [9E9, 9E9, 9E9, 9E9, 9E9, 9E9]];
	VAR jointtarget CDP_3156 := [[-12.15, 36.22, 5.26, 0, 48.52, 114.05], [9E9, 9E9, 9E9, 9E9, 9E9, 9E9]];
	VAR jointtarget CDP_3157 := [[-12.19, 36.19, 5.3, 0, 48.51, 116.2], [9E9, 9E9, 9E9, 9E9, 9E9, 9E9]];
	VAR jointtarget CDP_3158 := [[-12.24, 36.16, 5.35, 0, 48.49, 118.34], [9E9, 9E9, 9E9, 9E9, 9E9, 9E9]];
	VAR jointtarget CDP_3159 := [[-12.29, 36.13, 5.4, 0, 48.46, 120.49], [9E9, 9E9, 9E9, 9E9, 9E9, 9E9]];
	VAR jointtarget CDP_3160 := [[-12.32, 36.11, 5.44, 0, 48.45, 121.56], [9E9, 9E9, 9E9, 9E9, 9E9, 9E9]];
	VAR jointtarget CDP_3161 := [[-12.35, 36.09, 5.47, 0, 48.44, 121.53], [9E9, 9E9, 9E9, 9E9, 9E9, 9E9]];
	VAR jointtarget CDP_3162 := [[-12.38, 36.07, 5.5, 0, 48.42, 121.5], [9E9, 9E9, 9E9, 9E9, 9E9, 9E9]];
	VAR jointtarget CDP_3163 := [[-12.41, 36.06, 5.54, 0, 48.41, 121.47], [9E9, 9E9, 9E9, 9E9, 9E9, 9E9]];
	VAR jointtarget CDP_3164 := [[-12.43, 36.04, 5.57, 0, 48.4, 121.44], [9E9, 9E9, 9E9, 9E9, 9E9, 9E9]];
	VAR jointtarget CDP_3165 := [[-12.46, 36.02, 5.6, 0, 48.38, 121.41], [9E9, 9E9, 9E9, 9E9, 9E9, 9E9]];
	VAR jointtarget CDP_3166 := [[-12.49, 36, 5.63, 0, 48.37, 121.39], [9E9, 9E9, 9E9, 9E9, 9E9, 9E9]];
	VAR jointtarget CDP_3167 := [[-12.52, 35.98, 5.67, 0, 48.35, 121.36], [9E9, 9E9, 9E9, 9E9, 9E9, 9E9]];
	VAR jointtarget CDP_3168 := [[-12.55, 35.96, 5.7, 0, 48.34, 121.33], [9E9, 9E9, 9E9, 9E9, 9E9, 9E9]];
	VAR jointtarget CDP_3169 := [[-12.58, 35.94, 5.73, 0, 48.33, 121.3], [9E9, 9E9, 9E9, 9E9, 9E9, 9E9]];
	VAR jointtarget CDP_3170 := [[-12.61, 35.92, 5.76, 0, 48.31, 121.27], [9E9, 9E9, 9E9, 9E9, 9E9, 9E9]];
	VAR jointtarget CDP_3171 := [[-12.63, 35.9, 5.8, 0, 48.3, 121.24], [9E9, 9E9, 9E9, 9E9, 9E9, 9E9]];
	VAR jointtarget CDP_3172 := [[-12.66, 35.88, 5.83, 0, 48.29, 121.21], [9E9, 9E9, 9E9, 9E9, 9E9, 9E9]];
	VAR jointtarget CDP_3173 := [[-12.69, 35.87, 5.86, 0, 48.27, 121.18], [9E9, 9E9, 9E9, 9E9, 9E9, 9E9]];
	VAR jointtarget CDP_3174 := [[-12.72, 35.85, 5.89, 0, 48.26, 121.16], [9E9, 9E9, 9E9, 9E9, 9E9, 9E9]];
	VAR jointtarget CDP_3175 := [[-12.75, 35.83, 5.93, 0, 48.25, 121.13], [9E9, 9E9, 9E9, 9E9, 9E9, 9E9]];
	VAR jointtarget CDP_3176 := [[-12.78, 35.81, 5.96, 0, 48.23, 121.1], [9E9, 9E9, 9E9, 9E9, 9E9, 9E9]];
	VAR jointtarget CDP_3177 := [[-12.81, 35.79, 5.99, 0, 48.22, 121.07], [9E9, 9E9, 9E9, 9E9, 9E9, 9E9]];
	VAR jointtarget CDP_3178 := [[-12.84, 35.77, 6.02, 0, 48.21, 121.04], [9E9, 9E9, 9E9, 9E9, 9E9, 9E9]];
	VAR jointtarget CDP_3179 := [[-12.86, 35.75, 6.05, 0, 48.19, 121.01], [9E9, 9E9, 9E9, 9E9, 9E9, 9E9]];
	VAR jointtarget CDP_3180 := [[-13.02, 35.68, 6.18, 0, 48.14, 114.17], [9E9, 9E9, 9E9, 9E9, 9E9, 9E9]];
	VAR jointtarget CDP_3181 := [[-13.18, 35.65, 6.24, 0, 48.12, 100.62], [9E9, 9E9, 9E9, 9E9, 9E9, 9E9]];
	VAR jointtarget CDP_3182 := [[-13.34, 35.66, 6.22, 0, 48.12, 87.07], [9E9, 9E9, 9E9, 9E9, 9E9, 9E9]];
	VAR jointtarget CDP_3183 := [[-13.5, 35.71, 6.13, 0, 48.16, 73.52], [9E9, 9E9, 9E9, 9E9, 9E9, 9E9]];
	VAR jointtarget CDP_3184 := [[-13.64, 35.79, 5.98, 0, 48.22, 59.99], [9E9, 9E9, 9E9, 9E9, 9E9, 9E9]];
	VAR jointtarget CDP_3185 := [[-13.76, 35.92, 5.77, 0, 48.31, 46.48], [9E9, 9E9, 9E9, 9E9, 9E9, 9E9]];
	VAR jointtarget CDP_3186 := [[-13.85, 36.07, 5.52, 0, 48.42, 33.01], [9E9, 9E9, 9E9, 9E9, 9E9, 9E9]];
	VAR jointtarget CDP_3187 := [[-13.91, 36.24, 5.23, 0, 48.54, 19.56], [9E9, 9E9, 9E9, 9E9, 9E9, 9E9]];
	VAR jointtarget CDP_3188 := [[-13.92, 36.41, 4.92, 0, 48.66, 6.16], [9E9, 9E9, 9E9, 9E9, 9E9, 9E9]];
	VAR jointtarget CDP_3189 := [[-13.9, 36.59, 4.62, 0, 48.79, -7.21], [9E9, 9E9, 9E9, 9E9, 9E9, 9E9]];
	VAR jointtarget CDP_3190 := [[-13.85, 36.76, 4.33, 0, 48.91, -20.54], [9E9, 9E9, 9E9, 9E9, 9E9, 9E9]];
	VAR jointtarget CDP_3191 := [[-13.76, 36.91, 4.07, 0, 49.02, -33.84], [9E9, 9E9, 9E9, 9E9, 9E9, 9E9]];
	VAR jointtarget CDP_3192 := [[-13.64, 37.03, 3.86, 0, 49.11, -47.11], [9E9, 9E9, 9E9, 9E9, 9E9, 9E9]];
	VAR jointtarget CDP_3193 := [[-13.5, 37.12, 3.71, 0, 49.17, -60.35], [9E9, 9E9, 9E9, 9E9, 9E9, 9E9]];
	VAR jointtarget CDP_3194 := [[-13.34, 37.17, 3.62, 0, 49.21, -73.59], [9E9, 9E9, 9E9, 9E9, 9E9, 9E9]];
	VAR jointtarget CDP_3195 := [[-13.18, 37.18, 3.6, 0, 49.22, -86.81], [9E9, 9E9, 9E9, 9E9, 9E9, 9E9]];
	VAR jointtarget CDP_3196 := [[-13.02, 37.15, 3.66, 0, 49.19, -100.04], [9E9, 9E9, 9E9, 9E9, 9E9, 9E9]];
	VAR jointtarget CDP_3197 := [[-12.88, 37.08, 3.78, 0, 49.14, -113.28], [9E9, 9E9, 9E9, 9E9, 9E9, 9E9]];
	VAR jointtarget CDP_3198 := [[-12.75, 36.97, 3.96, 0, 49.07, -126.54], [9E9, 9E9, 9E9, 9E9, 9E9, 9E9]];
	VAR jointtarget CDP_3199 := [[-12.64, 36.83, 4.2, 0, 48.97, -139.82], [9E9, 9E9, 9E9, 9E9, 9E9, 9E9]];
	VAR jointtarget CDP_3200 := [[-12.62, 36.79, 4.27, 0, 48.94, -146.49], [9E9, 9E9, 9E9, 9E9, 9E9, 9E9]];
	VAR jointtarget CDP_3201 := [[-12.59, 36.75, 4.34, 0, 48.91, -146.47], [9E9, 9E9, 9E9, 9E9, 9E9, 9E9]];
	VAR jointtarget CDP_3202 := [[-12.57, 36.71, 4.41, 0, 48.88, -146.44], [9E9, 9E9, 9E9, 9E9, 9E9, 9E9]];
	VAR jointtarget CDP_3203 := [[-12.54, 36.67, 4.49, 0, 48.85, -146.42], [9E9, 9E9, 9E9, 9E9, 9E9, 9E9]];
	VAR jointtarget CDP_3204 := [[-12.52, 36.63, 4.56, 0, 48.82, -146.4], [9E9, 9E9, 9E9, 9E9, 9E9, 9E9]];
	VAR jointtarget CDP_3205 := [[-12.49, 36.59, 4.63, 0, 48.79, -146.37], [9E9, 9E9, 9E9, 9E9, 9E9, 9E9]];
	VAR jointtarget CDP_3206 := [[-12.47, 36.54, 4.7, 0, 48.76, -146.35], [9E9, 9E9, 9E9, 9E9, 9E9, 9E9]];
	VAR jointtarget CDP_3207 := [[-12.44, 36.5, 4.77, 0, 48.73, -146.32], [9E9, 9E9, 9E9, 9E9, 9E9, 9E9]];
	VAR jointtarget CDP_3208 := [[-12.42, 36.46, 4.84, 0, 48.7, -146.3], [9E9, 9E9, 9E9, 9E9, 9E9, 9E9]];
	VAR jointtarget CDP_3209 := [[-12.39, 36.42, 4.91, 0, 48.67, -146.27], [9E9, 9E9, 9E9, 9E9, 9E9, 9E9]];
	VAR jointtarget CDP_3210 := [[-12.37, 36.38, 4.98, 0, 48.64, -146.25], [9E9, 9E9, 9E9, 9E9, 9E9, 9E9]];
	VAR jointtarget CDP_3211 := [[-12.34, 36.34, 5.05, 0, 48.61, -146.22], [9E9, 9E9, 9E9, 9E9, 9E9, 9E9]];
	VAR jointtarget CDP_3212 := [[-12.32, 36.3, 5.12, 0, 48.58, -146.2], [9E9, 9E9, 9E9, 9E9, 9E9, 9E9]];
	VAR jointtarget CDP_3213 := [[-12.29, 36.26, 5.19, 0, 48.55, -146.17], [9E9, 9E9, 9E9, 9E9, 9E9, 9E9]];
	VAR jointtarget CDP_3214 := [[-12.27, 36.22, 5.26, 0, 48.52, -146.15], [9E9, 9E9, 9E9, 9E9, 9E9, 9E9]];
	VAR jointtarget CDP_3215 := [[-12.24, 36.18, 5.33, 0, 48.49, -146.12], [9E9, 9E9, 9E9, 9E9, 9E9, 9E9]];
	VAR jointtarget CDP_3216 := [[-12.22, 36.13, 5.4, 0, 48.46, -146.1], [9E9, 9E9, 9E9, 9E9, 9E9, 9E9]];
	VAR jointtarget CDP_3217 := [[-12.19, 36.09, 5.47, 0, 48.44, -146.07], [9E9, 9E9, 9E9, 9E9, 9E9, 9E9]];
	VAR jointtarget CDP_3218 := [[-12.17, 36.05, 5.54, 0, 48.41, -146.05], [9E9, 9E9, 9E9, 9E9, 9E9, 9E9]];
	VAR jointtarget CDP_3219 := [[-12.14, 36.01, 5.61, 0, 48.38, -146.02], [9E9, 9E9, 9E9, 9E9, 9E9, 9E9]];
	VAR jointtarget CDP_3220 := [[-12.14, 36, 5.63, 0, 48.37, -145.46], [9E9, 9E9, 9E9, 9E9, 9E9, 9E9]];
	VAR jointtarget CDP_3221 := [[-12.13, 35.99, 5.65, 0, 48.36, -144.35], [9E9, 9E9, 9E9, 9E9, 9E9, 9E9]];
	VAR jointtarget CDP_3222 := [[-12.12, 35.97, 5.67, 0, 48.35, -143.24], [9E9, 9E9, 9E9, 9E9, 9E9, 9E9]];
	VAR jointtarget CDP_3223 := [[-12.11, 35.96, 5.69, 0, 48.34, -142.13], [9E9, 9E9, 9E9, 9E9, 9E9, 9E9]];
	VAR jointtarget CDP_3224 := [[-12.1, 35.95, 5.72, 0, 48.33, -141.01], [9E9, 9E9, 9E9, 9E9, 9E9, 9E9]];
	VAR jointtarget CDP_3225 := [[-12.09, 35.94, 5.74, 0, 48.33, -139.9], [9E9, 9E9, 9E9, 9E9, 9E9, 9E9]];
	VAR jointtarget CDP_3226 := [[-12.08, 35.93, 5.75, 0, 48.32, -138.79], [9E9, 9E9, 9E9, 9E9, 9E9, 9E9]];
	VAR jointtarget CDP_3227 := [[-12.07, 35.92, 5.77, 0, 48.31, -137.68], [9E9, 9E9, 9E9, 9E9, 9E9, 9E9]];
	VAR jointtarget CDP_3228 := [[-12.06, 35.9, 5.79, 0, 48.3, -136.56], [9E9, 9E9, 9E9, 9E9, 9E9, 9E9]];
	VAR jointtarget CDP_3229 := [[-12.05, 35.89, 5.81, 0, 48.3, -135.45], [9E9, 9E9, 9E9, 9E9, 9E9, 9E9]];
	VAR jointtarget CDP_3230 := [[-12.04, 35.88, 5.83, 0, 48.29, -134.34], [9E9, 9E9, 9E9, 9E9, 9E9, 9E9]];
	VAR jointtarget CDP_3231 := [[-12.03, 35.87, 5.85, 0, 48.28, -133.22], [9E9, 9E9, 9E9, 9E9, 9E9, 9E9]];
	VAR jointtarget CDP_3232 := [[-12.02, 35.86, 5.87, 0, 48.27, -132.11], [9E9, 9E9, 9E9, 9E9, 9E9, 9E9]];
	VAR jointtarget CDP_3233 := [[-12.01, 35.85, 5.88, 0, 48.27, -130.99], [9E9, 9E9, 9E9, 9E9, 9E9, 9E9]];
	VAR jointtarget CDP_3234 := [[-12, 35.84, 5.9, 0, 48.26, -129.88], [9E9, 9E9, 9E9, 9E9, 9E9, 9E9]];
	VAR jointtarget CDP_3235 := [[-11.99, 35.83, 5.91, 0, 48.25, -128.76], [9E9, 9E9, 9E9, 9E9, 9E9, 9E9]];
	VAR jointtarget CDP_3236 := [[-11.98, 35.82, 5.93, 0, 48.25, -127.65], [9E9, 9E9, 9E9, 9E9, 9E9, 9E9]];
	VAR jointtarget CDP_3237 := [[-11.97, 35.81, 5.95, 0, 48.24, -126.53], [9E9, 9E9, 9E9, 9E9, 9E9, 9E9]];
	VAR jointtarget CDP_3238 := [[-11.96, 35.8, 5.96, 0, 48.24, -125.42], [9E9, 9E9, 9E9, 9E9, 9E9, 9E9]];
	VAR jointtarget CDP_3239 := [[-11.95, 35.79, 5.98, 0, 48.23, -124.3], [9E9, 9E9, 9E9, 9E9, 9E9, 9E9]];
	VAR jointtarget CDP_3240 := [[-11.94, 35.79, 5.99, 0, 48.23, -123.74], [9E9, 9E9, 9E9, 9E9, 9E9, 9E9]];
	VAR jointtarget CDP_3241 := [[-11.93, 35.78, 6, 0, 48.22, -123.73], [9E9, 9E9, 9E9, 9E9, 9E9, 9E9]];
	VAR jointtarget CDP_3242 := [[-11.92, 35.77, 6.01, 0, 48.22, -123.72], [9E9, 9E9, 9E9, 9E9, 9E9, 9E9]];
	VAR jointtarget CDP_3243 := [[-11.9, 35.76, 6.03, 0, 48.21, -123.71], [9E9, 9E9, 9E9, 9E9, 9E9, 9E9]];
	VAR jointtarget CDP_3244 := [[-11.89, 35.75, 6.04, 0, 48.21, -123.7], [9E9, 9E9, 9E9, 9E9, 9E9, 9E9]];
	VAR jointtarget CDP_3245 := [[-11.88, 35.75, 6.05, 0, 48.2, -123.69], [9E9, 9E9, 9E9, 9E9, 9E9, 9E9]];
	VAR jointtarget CDP_3246 := [[-11.87, 35.74, 6.06, 0, 48.2, -123.68], [9E9, 9E9, 9E9, 9E9, 9E9, 9E9]];
	VAR jointtarget CDP_3247 := [[-11.86, 35.73, 6.08, 0, 48.19, -123.66], [9E9, 9E9, 9E9, 9E9, 9E9, 9E9]];
	VAR jointtarget CDP_3248 := [[-11.85, 35.72, 6.09, 0, 48.19, -123.65], [9E9, 9E9, 9E9, 9E9, 9E9, 9E9]];
	VAR jointtarget CDP_3249 := [[-11.84, 35.71, 6.1, 0, 48.18, -123.64], [9E9, 9E9, 9E9, 9E9, 9E9, 9E9]];
	VAR jointtarget CDP_3250 := [[-11.83, 35.71, 6.12, 0, 48.18, -123.63], [9E9, 9E9, 9E9, 9E9, 9E9, 9E9]];
	VAR jointtarget CDP_3251 := [[-11.82, 35.7, 6.13, 0, 48.17, -123.62], [9E9, 9E9, 9E9, 9E9, 9E9, 9E9]];
	VAR jointtarget CDP_3252 := [[-11.81, 35.69, 6.14, 0, 48.17, -123.61], [9E9, 9E9, 9E9, 9E9, 9E9, 9E9]];
	VAR jointtarget CDP_3253 := [[-11.8, 35.68, 6.15, 0, 48.16, -123.6], [9E9, 9E9, 9E9, 9E9, 9E9, 9E9]];
	VAR jointtarget CDP_3254 := [[-11.79, 35.67, 6.17, 0, 48.16, -123.59], [9E9, 9E9, 9E9, 9E9, 9E9, 9E9]];
	VAR jointtarget CDP_3255 := [[-11.78, 35.67, 6.18, 0, 48.15, -123.58], [9E9, 9E9, 9E9, 9E9, 9E9, 9E9]];
	VAR jointtarget CDP_3256 := [[-11.77, 35.66, 6.19, 0, 48.15, -123.57], [9E9, 9E9, 9E9, 9E9, 9E9, 9E9]];
	VAR jointtarget CDP_3257 := [[-11.76, 35.65, 6.2, 0, 48.14, -123.56], [9E9, 9E9, 9E9, 9E9, 9E9, 9E9]];
	VAR jointtarget CDP_3258 := [[-11.75, 35.64, 6.22, 0, 48.14, -123.55], [9E9, 9E9, 9E9, 9E9, 9E9, 9E9]];
	VAR jointtarget CDP_3259 := [[-11.74, 35.64, 6.23, 0, 48.13, -123.54], [9E9, 9E9, 9E9, 9E9, 9E9, 9E9]];
	VAR jointtarget CDP_3260 := [[-10.65, 35.4, 6.63, 0, 47.97, -100.65], [9E9, 9E9, 9E9, 9E9, 9E9, 9E9]];
	VAR jointtarget CDP_3261 := [[-9.55, 35.19, 6.98, 0, 47.82, -99.55], [9E9, 9E9, 9E9, 9E9, 9E9, 9E9]];
	VAR jointtarget CDP_3262 := [[-8.44, 35.01, 7.3, 0, 47.69, -98.44], [9E9, 9E9, 9E9, 9E9, 9E9, 9E9]];
	VAR jointtarget CDP_3263 := [[-7.33, 34.84, 7.58, 0, 47.58, -97.33], [9E9, 9E9, 9E9, 9E9, 9E9, 9E9]];
	VAR jointtarget CDP_3264 := [[-6.21, 34.7, 7.82, 0, 47.48, -96.21], [9E9, 9E9, 9E9, 9E9, 9E9, 9E9]];
	VAR jointtarget CDP_3265 := [[-5.09, 34.59, 8.02, 0, 47.4, -95.09], [9E9, 9E9, 9E9, 9E9, 9E9, 9E9]];
	VAR jointtarget CDP_3266 := [[-3.96, 34.49, 8.18, 0, 47.33, -93.96], [9E9, 9E9, 9E9, 9E9, 9E9, 9E9]];
	VAR jointtarget CDP_3267 := [[-2.83, 34.42, 8.3, 0, 47.28, -92.83], [9E9, 9E9, 9E9, 9E9, 9E9, 9E9]];
	VAR jointtarget CDP_3268 := [[-1.7, 34.37, 8.38, 0, 47.25, -91.7], [9E9, 9E9, 9E9, 9E9, 9E9, 9E9]];
	VAR jointtarget CDP_3269 := [[-0.56, 34.35, 8.42, 0, 47.23, -90.56], [9E9, 9E9, 9E9, 9E9, 9E9, 9E9]];
	VAR jointtarget CDP_3270 := [[0.57, 34.35, 8.42, 0, 47.23, -89.43], [9E9, 9E9, 9E9, 9E9, 9E9, 9E9]];
	VAR jointtarget CDP_3271 := [[1.7, 34.37, 8.38, 0, 47.25, -88.3], [9E9, 9E9, 9E9, 9E9, 9E9, 9E9]];
	VAR jointtarget CDP_3272 := [[2.84, 34.42, 8.3, 0, 47.28, -87.16], [9E9, 9E9, 9E9, 9E9, 9E9, 9E9]];
	VAR jointtarget CDP_3273 := [[3.97, 34.49, 8.18, 0, 47.33, -86.03], [9E9, 9E9, 9E9, 9E9, 9E9, 9E9]];
	VAR jointtarget CDP_3274 := [[5.09, 34.59, 8.02, 0, 47.4, -84.91], [9E9, 9E9, 9E9, 9E9, 9E9, 9E9]];
	VAR jointtarget CDP_3275 := [[6.22, 34.7, 7.82, 0, 47.48, -83.78], [9E9, 9E9, 9E9, 9E9, 9E9, 9E9]];
	VAR jointtarget CDP_3276 := [[7.34, 34.84, 7.58, 0, 47.58, -82.66], [9E9, 9E9, 9E9, 9E9, 9E9, 9E9]];
	VAR jointtarget CDP_3277 := [[8.45, 35.01, 7.3, 0, 47.69, -81.55], [9E9, 9E9, 9E9, 9E9, 9E9, 9E9]];
	VAR jointtarget CDP_3278 := [[9.56, 35.19, 6.98, 0, 47.82, -80.44], [9E9, 9E9, 9E9, 9E9, 9E9, 9E9]];
	VAR jointtarget CDP_3279 := [[10.65, 35.4, 6.62, 0, 47.97, -79.35], [9E9, 9E9, 9E9, 9E9, 9E9, 9E9]];
	VAR jointtarget CDP_3280 := [[10.71, 35.42, 6.6, 0, 47.98, -78.19], [9E9, 9E9, 9E9, 9E9, 9E9, 9E9]];
	VAR jointtarget CDP_3281 := [[10.76, 35.43, 6.58, 0, 47.99, -75.95], [9E9, 9E9, 9E9, 9E9, 9E9, 9E9]];
	VAR jointtarget CDP_3282 := [[10.82, 35.45, 6.55, 0, 48, -73.7], [9E9, 9E9, 9E9, 9E9, 9E9, 9E9]];
	VAR jointtarget CDP_3283 := [[10.87, 35.47, 6.52, 0, 48.02, -71.45], [9E9, 9E9, 9E9, 9E9, 9E9, 9E9]];
	VAR jointtarget CDP_3284 := [[10.92, 35.49, 6.48, 0, 48.03, -69.2], [9E9, 9E9, 9E9, 9E9, 9E9, 9E9]];
	VAR jointtarget CDP_3285 := [[10.97, 35.51, 6.44, 0, 48.05, -66.96], [9E9, 9E9, 9E9, 9E9, 9E9, 9E9]];
	VAR jointtarget CDP_3286 := [[11.03, 35.54, 6.4, 0, 48.07, -64.72], [9E9, 9E9, 9E9, 9E9, 9E9, 9E9]];
	VAR jointtarget CDP_3287 := [[11.07, 35.57, 6.35, 0, 48.09, -62.47], [9E9, 9E9, 9E9, 9E9, 9E9, 9E9]];
	VAR jointtarget CDP_3288 := [[11.12, 35.6, 6.3, 0, 48.11, -60.23], [9E9, 9E9, 9E9, 9E9, 9E9, 9E9]];
	VAR jointtarget CDP_3289 := [[11.17, 35.63, 6.24, 0, 48.13, -57.99], [9E9, 9E9, 9E9, 9E9, 9E9, 9E9]];
	VAR jointtarget CDP_3290 := [[11.22, 35.66, 6.19, 0, 48.15, -55.75], [9E9, 9E9, 9E9, 9E9, 9E9, 9E9]];
	VAR jointtarget CDP_3291 := [[11.26, 35.7, 6.12, 0, 48.18, -53.51], [9E9, 9E9, 9E9, 9E9, 9E9, 9E9]];
	VAR jointtarget CDP_3292 := [[11.3, 35.73, 6.06, 0, 48.21, -51.27], [9E9, 9E9, 9E9, 9E9, 9E9, 9E9]];
	VAR jointtarget CDP_3293 := [[11.35, 35.77, 5.99, 0, 48.23, -49.04], [9E9, 9E9, 9E9, 9E9, 9E9, 9E9]];
	VAR jointtarget CDP_3294 := [[11.39, 35.82, 5.92, 0, 48.26, -46.8], [9E9, 9E9, 9E9, 9E9, 9E9, 9E9]];
	VAR jointtarget CDP_3295 := [[11.43, 35.86, 5.85, 0, 48.29, -44.57], [9E9, 9E9, 9E9, 9E9, 9E9, 9E9]];
	VAR jointtarget CDP_3296 := [[11.46, 35.9, 5.77, 0, 48.32, -42.34], [9E9, 9E9, 9E9, 9E9, 9E9, 9E9]];
	VAR jointtarget CDP_3297 := [[11.5, 35.95, 5.69, 0, 48.36, -40.11], [9E9, 9E9, 9E9, 9E9, 9E9, 9E9]];
	VAR jointtarget CDP_3298 := [[11.53, 36, 5.61, 0, 48.39, -37.88], [9E9, 9E9, 9E9, 9E9, 9E9, 9E9]];
	VAR jointtarget CDP_3299 := [[11.57, 36.05, 5.53, 0, 48.43, -35.65], [9E9, 9E9, 9E9, 9E9, 9E9, 9E9]];
	VAR jointtarget CDP_3300 := [[11.59, 36.08, 5.48, 0, 48.45, -34.54], [9E9, 9E9, 9E9, 9E9, 9E9, 9E9]];
	VAR jointtarget CDP_3301 := [[11.6, 36.11, 5.42, 0, 48.47, -34.52], [9E9, 9E9, 9E9, 9E9, 9E9, 9E9]];
	VAR jointtarget CDP_3302 := [[11.62, 36.14, 5.37, 0, 48.49, -34.5], [9E9, 9E9, 9E9, 9E9, 9E9, 9E9]];
	VAR jointtarget CDP_3303 := [[11.64, 36.17, 5.32, 0, 48.51, -34.48], [9E9, 9E9, 9E9, 9E9, 9E9, 9E9]];
	VAR jointtarget CDP_3304 := [[11.66, 36.2, 5.27, 0, 48.53, -34.46], [9E9, 9E9, 9E9, 9E9, 9E9, 9E9]];
	VAR jointtarget CDP_3305 := [[11.68, 36.23, 5.22, 0, 48.56, -34.44], [9E9, 9E9, 9E9, 9E9, 9E9, 9E9]];
	VAR jointtarget CDP_3306 := [[11.7, 36.26, 5.17, 0, 48.58, -34.42], [9E9, 9E9, 9E9, 9E9, 9E9, 9E9]];
	VAR jointtarget CDP_3307 := [[11.72, 36.29, 5.11, 0, 48.6, -34.41], [9E9, 9E9, 9E9, 9E9, 9E9, 9E9]];
	VAR jointtarget CDP_3308 := [[11.74, 36.32, 5.06, 0, 48.62, -34.39], [9E9, 9E9, 9E9, 9E9, 9E9, 9E9]];
	VAR jointtarget CDP_3309 := [[11.76, 36.35, 5.01, 0, 48.64, -34.37], [9E9, 9E9, 9E9, 9E9, 9E9, 9E9]];
	VAR jointtarget CDP_3310 := [[11.77, 36.38, 4.96, 0, 48.66, -34.35], [9E9, 9E9, 9E9, 9E9, 9E9, 9E9]];
	VAR jointtarget CDP_3311 := [[11.79, 36.41, 4.91, 0, 48.69, -34.33], [9E9, 9E9, 9E9, 9E9, 9E9, 9E9]];
	VAR jointtarget CDP_3312 := [[11.81, 36.44, 4.85, 0, 48.71, -34.31], [9E9, 9E9, 9E9, 9E9, 9E9, 9E9]];
	VAR jointtarget CDP_3313 := [[11.83, 36.47, 4.8, 0, 48.73, -34.29], [9E9, 9E9, 9E9, 9E9, 9E9, 9E9]];
	VAR jointtarget CDP_3314 := [[11.85, 36.5, 4.75, 0, 48.75, -34.27], [9E9, 9E9, 9E9, 9E9, 9E9, 9E9]];
	VAR jointtarget CDP_3315 := [[11.87, 36.53, 4.7, 0, 48.77, -34.26], [9E9, 9E9, 9E9, 9E9, 9E9, 9E9]];
	VAR jointtarget CDP_3316 := [[11.89, 36.56, 4.65, 0, 48.79, -34.24], [9E9, 9E9, 9E9, 9E9, 9E9, 9E9]];
	VAR jointtarget CDP_3317 := [[11.91, 36.59, 4.59, 0, 48.82, -34.22], [9E9, 9E9, 9E9, 9E9, 9E9, 9E9]];
	VAR jointtarget CDP_3318 := [[11.92, 36.62, 4.54, 0, 48.84, -34.2], [9E9, 9E9, 9E9, 9E9, 9E9, 9E9]];
	VAR jointtarget CDP_3319 := [[11.94, 36.65, 4.49, 0, 48.86, -34.18], [9E9, 9E9, 9E9, 9E9, 9E9, 9E9]];
	VAR jointtarget CDP_3320 := [[12.05, 36.79, 4.26, 0, 48.96, -40.77], [9E9, 9E9, 9E9, 9E9, 9E9, 9E9]];
	VAR jointtarget CDP_3321 := [[12.18, 36.89, 4.07, 0, 49.03, -54.03], [9E9, 9E9, 9E9, 9E9, 9E9, 9E9]];
	VAR jointtarget CDP_3322 := [[12.33, 36.96, 3.96, 0, 49.08, -67.26], [9E9, 9E9, 9E9, 9E9, 9E9, 9E9]];
	VAR jointtarget CDP_3323 := [[12.49, 36.99, 3.9, 0, 49.1, -80.49], [9E9, 9E9, 9E9, 9E9, 9E9, 9E9]];
	VAR jointtarget CDP_3324 := [[12.65, 36.98, 3.92, 0, 49.1, -93.72], [9E9, 9E9, 9E9, 9E9, 9E9, 9E9]];
	VAR jointtarget CDP_3325 := [[12.8, 36.93, 4.02, 0, 49.06, -106.95], [9E9, 9E9, 9E9, 9E9, 9E9, 9E9]];
	VAR jointtarget CDP_3326 := [[12.94, 36.84, 4.17, 0, 48.99, -120.2], [9E9, 9E9, 9E9, 9E9, 9E9, 9E9]];
	VAR jointtarget CDP_3327 := [[13.06, 36.71, 4.38, 0, 48.9, -133.47], [9E9, 9E9, 9E9, 9E9, 9E9, 9E9]];
	VAR jointtarget CDP_3328 := [[13.15, 36.56, 4.64, 0, 48.8, -146.77], [9E9, 9E9, 9E9, 9E9, 9E9, 9E9]];
	VAR jointtarget CDP_3329 := [[13.2, 36.39, 4.93, 0, 48.67, -160.1], [9E9, 9E9, 9E9, 9E9, 9E9, 9E9]];
	VAR jointtarget CDP_3330 := [[13.22, 36.21, 5.24, 0, 48.55, -173.47], [9E9, 9E9, 9E9, 9E9, 9E9, 9E9]];
	VAR jointtarget CDP_3331 := [[13.2, 36.04, 5.54, 0, 48.42, -186.88], [9E9, 9E9, 9E9, 9E9, 9E9, 9E9]];
	VAR jointtarget CDP_3332 := [[13.15, 35.87, 5.83, 0, 48.3, -200.32], [9E9, 9E9, 9E9, 9E9, 9E9, 9E9]];
	VAR jointtarget CDP_3333 := [[13.06, 35.72, 6.08, 0, 48.2, -213.8], [9E9, 9E9, 9E9, 9E9, 9E9, 9E9]];
	VAR jointtarget CDP_3334 := [[12.93, 35.6, 6.29, 0, 48.11, -227.31], [9E9, 9E9, 9E9, 9E9, 9E9, 9E9]];
	VAR jointtarget CDP_3335 := [[12.79, 35.51, 6.44, 0, 48.05, -240.84], [9E9, 9E9, 9E9, 9E9, 9E9, 9E9]];
	VAR jointtarget CDP_3336 := [[12.63, 35.47, 6.52, 0, 48.01, -254.39], [9E9, 9E9, 9E9, 9E9, 9E9, 9E9]];
	VAR jointtarget CDP_3337 := [[12.47, 35.46, 6.53, 0, 48.01, -267.94], [9E9, 9E9, 9E9, 9E9, 9E9, 9E9]];
	VAR jointtarget CDP_3338 := [[12.3, 35.49, 6.47, 0, 48.03, -281.49], [9E9, 9E9, 9E9, 9E9, 9E9, 9E9]];
	VAR jointtarget CDP_3339 := [[12.15, 35.57, 6.34, 0, 48.09, -295.03], [9E9, 9E9, 9E9, 9E9, 9E9, 9E9]];
	VAR jointtarget CDP_3340 := [[12.13, 35.59, 6.31, 0, 48.1, -301.75], [9E9, 9E9, 9E9, 9E9, 9E9, 9E9]];
	VAR jointtarget CDP_3341 := [[12.1, 35.61, 6.28, 0, 48.12, -301.78], [9E9, 9E9, 9E9, 9E9, 9E9, 9E9]];
	VAR jointtarget CDP_3342 := [[12.07, 35.63, 6.24, 0, 48.13, -301.81], [9E9, 9E9, 9E9, 9E9, 9E9, 9E9]];
	VAR jointtarget CDP_3343 := [[12.04, 35.65, 6.21, 0, 48.14, -301.84], [9E9, 9E9, 9E9, 9E9, 9E9, 9E9]];
	VAR jointtarget CDP_3344 := [[12.01, 35.67, 6.18, 0, 48.16, -301.87], [9E9, 9E9, 9E9, 9E9, 9E9, 9E9]];
	VAR jointtarget CDP_3345 := [[11.98, 35.68, 6.15, 0, 48.17, -301.89], [9E9, 9E9, 9E9, 9E9, 9E9, 9E9]];
	VAR jointtarget CDP_3346 := [[11.95, 35.7, 6.11, 0, 48.18, -301.92], [9E9, 9E9, 9E9, 9E9, 9E9, 9E9]];
	VAR jointtarget CDP_3347 := [[11.92, 35.72, 6.08, 0, 48.2, -301.95], [9E9, 9E9, 9E9, 9E9, 9E9, 9E9]];
	VAR jointtarget CDP_3348 := [[11.9, 35.74, 6.05, 0, 48.21, -301.98], [9E9, 9E9, 9E9, 9E9, 9E9, 9E9]];
	VAR jointtarget CDP_3349 := [[11.87, 35.76, 6.01, 0, 48.22, -302.01], [9E9, 9E9, 9E9, 9E9, 9E9, 9E9]];
	VAR jointtarget CDP_3350 := [[11.84, 35.78, 5.98, 0, 48.24, -302.04], [9E9, 9E9, 9E9, 9E9, 9E9, 9E9]];
	VAR jointtarget CDP_3351 := [[11.81, 35.8, 5.95, 0, 48.25, -302.07], [9E9, 9E9, 9E9, 9E9, 9E9, 9E9]];
	VAR jointtarget CDP_3352 := [[11.78, 35.82, 5.91, 0, 48.27, -302.09], [9E9, 9E9, 9E9, 9E9, 9E9, 9E9]];
	VAR jointtarget CDP_3353 := [[11.75, 35.84, 5.88, 0, 48.28, -302.12], [9E9, 9E9, 9E9, 9E9, 9E9, 9E9]];
	VAR jointtarget CDP_3354 := [[11.73, 35.86, 5.85, 0, 48.29, -302.15], [9E9, 9E9, 9E9, 9E9, 9E9, 9E9]];
	VAR jointtarget CDP_3355 := [[11.7, 35.88, 5.82, 0, 48.31, -302.18], [9E9, 9E9, 9E9, 9E9, 9E9, 9E9]];
	VAR jointtarget CDP_3356 := [[11.67, 35.9, 5.78, 0, 48.32, -302.21], [9E9, 9E9, 9E9, 9E9, 9E9, 9E9]];
	VAR jointtarget CDP_3357 := [[11.64, 35.92, 5.75, 0, 48.33, -302.24], [9E9, 9E9, 9E9, 9E9, 9E9, 9E9]];
	VAR jointtarget CDP_3358 := [[11.61, 35.94, 5.72, 0, 48.35, -302.27], [9E9, 9E9, 9E9, 9E9, 9E9, 9E9]];
	VAR jointtarget CDP_3359 := [[11.58, 35.96, 5.68, 0, 48.36, -302.29], [9E9, 9E9, 9E9, 9E9, 9E9, 9E9]];
	VAR jointtarget CDP_3360 := [[11.54, 35.99, 5.63, 0, 48.38, -301.24], [9E9, 9E9, 9E9, 9E9, 9E9, 9E9]];
	VAR jointtarget CDP_3361 := [[11.49, 36.02, 5.58, 0, 48.41, -299.1], [9E9, 9E9, 9E9, 9E9, 9E9, 9E9]];
	VAR jointtarget CDP_3362 := [[11.44, 36.04, 5.53, 0, 48.43, -296.95], [9E9, 9E9, 9E9, 9E9, 9E9, 9E9]];
	VAR jointtarget CDP_3363 := [[11.39, 36.07, 5.49, 0, 48.44, -294.81], [9E9, 9E9, 9E9, 9E9, 9E9, 9E9]];
	VAR jointtarget CDP_3364 := [[11.34, 36.09, 5.45, 0, 48.46, -292.67], [9E9, 9E9, 9E9, 9E9, 9E9, 9E9]];
	VAR jointtarget CDP_3365 := [[11.28, 36.11, 5.41, 0, 48.47, -290.53], [9E9, 9E9, 9E9, 9E9, 9E9, 9E9]];
	VAR jointtarget CDP_3366 := [[11.23, 36.13, 5.38, 0, 48.49, -288.38], [9E9, 9E9, 9E9, 9E9, 9E9, 9E9]];
	VAR jointtarget CDP_3367 := [[11.18, 36.15, 5.35, 0, 48.5, -286.24], [9E9, 9E9, 9E9, 9E9, 9E9, 9E9]];
	VAR jointtarget CDP_3368 := [[11.13, 36.16, 5.32, 0, 48.51, -284.1], [9E9, 9E9, 9E9, 9E9, 9E9, 9E9]];
	VAR jointtarget CDP_3369 := [[11.07, 36.18, 5.3, 0, 48.52, -281.96], [9E9, 9E9, 9E9, 9E9, 9E9, 9E9]];
	VAR jointtarget CDP_3370 := [[11.02, 36.19, 5.29, 0, 48.53, -279.82], [9E9, 9E9, 9E9, 9E9, 9E9, 9E9]];
	VAR jointtarget CDP_3371 := [[10.96, 36.2, 5.27, 0, 48.53, -277.69], [9E9, 9E9, 9E9, 9E9, 9E9, 9E9]];
	VAR jointtarget CDP_3372 := [[10.91, 36.2, 5.26, 0, 48.54, -275.55], [9E9, 9E9, 9E9, 9E9, 9E9, 9E9]];
	VAR jointtarget CDP_3373 := [[10.85, 36.2, 5.26, 0, 48.54, -273.41], [9E9, 9E9, 9E9, 9E9, 9E9, 9E9]];
	VAR jointtarget CDP_3374 := [[10.8, 36.21, 5.25, 0, 48.54, -271.27], [9E9, 9E9, 9E9, 9E9, 9E9, 9E9]];
	VAR jointtarget CDP_3375 := [[10.74, 36.2, 5.26, 0, 48.54, -269.13], [9E9, 9E9, 9E9, 9E9, 9E9, 9E9]];
	VAR jointtarget CDP_3376 := [[10.69, 36.2, 5.26, 0, 48.54, -266.99], [9E9, 9E9, 9E9, 9E9, 9E9, 9E9]];
	VAR jointtarget CDP_3377 := [[10.63, 36.2, 5.27, 0, 48.53, -264.85], [9E9, 9E9, 9E9, 9E9, 9E9, 9E9]];
	VAR jointtarget CDP_3378 := [[10.58, 36.19, 5.28, 0, 48.53, -262.71], [9E9, 9E9, 9E9, 9E9, 9E9, 9E9]];
	VAR jointtarget CDP_3379 := [[10.52, 36.18, 5.3, 0, 48.52, -260.58], [9E9, 9E9, 9E9, 9E9, 9E9, 9E9]];
	VAR jointtarget CDP_3380 := [[9.44, 35.97, 5.65, 0, 48.37, -260.56], [9E9, 9E9, 9E9, 9E9, 9E9, 9E9]];
	VAR jointtarget CDP_3381 := [[8.36, 35.79, 5.97, 0, 48.24, -261.64], [9E9, 9E9, 9E9, 9E9, 9E9, 9E9]];
	VAR jointtarget CDP_3382 := [[7.27, 35.63, 6.25, 0, 48.13, -262.73], [9E9, 9E9, 9E9, 9E9, 9E9, 9E9]];
	VAR jointtarget CDP_3383 := [[6.17, 35.49, 6.48, 0, 48.03, -263.83], [9E9, 9E9, 9E9, 9E9, 9E9, 9E9]];
	VAR jointtarget CDP_3384 := [[5.07, 35.37, 6.68, 0, 47.95, -264.93], [9E9, 9E9, 9E9, 9E9, 9E9, 9E9]];
	VAR jointtarget CDP_3385 := [[3.97, 35.28, 6.84, 0, 47.88, -266.03], [9E9, 9E9, 9E9, 9E9, 9E9, 9E9]];
	VAR jointtarget CDP_3386 := [[2.86, 35.21, 6.96, 0, 47.83, -267.14], [9E9, 9E9, 9E9, 9E9, 9E9, 9E9]];
	VAR jointtarget CDP_3387 := [[1.75, 35.16, 7.04, 0, 47.8, -268.25], [9E9, 9E9, 9E9, 9E9, 9E9, 9E9]];
	VAR jointtarget CDP_3388 := [[0.64, 35.13, 7.09, 0, 47.78, -269.36], [9E9, 9E9, 9E9, 9E9, 9E9, 9E9]];
	VAR jointtarget CDP_3389 := [[-0.47, 35.13, 7.09, 0, 47.78, -270.47], [9E9, 9E9, 9E9, 9E9, 9E9, 9E9]];
	VAR jointtarget CDP_3390 := [[-1.58, 35.15, 7.05, 0, 47.79, -271.58], [9E9, 9E9, 9E9, 9E9, 9E9, 9E9]];
	VAR jointtarget CDP_3391 := [[-2.69, 35.2, 6.98, 0, 47.82, -272.69], [9E9, 9E9, 9E9, 9E9, 9E9, 9E9]];
	VAR jointtarget CDP_3392 := [[-3.8, 35.26, 6.86, 0, 47.87, -273.8], [9E9, 9E9, 9E9, 9E9, 9E9, 9E9]];
	VAR jointtarget CDP_3393 := [[-4.9, 35.35, 6.71, 0, 47.94, -274.9], [9E9, 9E9, 9E9, 9E9, 9E9, 9E9]];
	VAR jointtarget CDP_3394 := [[-6, 35.47, 6.52, 0, 48.02, -276], [9E9, 9E9, 9E9, 9E9, 9E9, 9E9]];
	VAR jointtarget CDP_3395 := [[-7.1, 35.6, 6.29, 0, 48.11, -277.1], [9E9, 9E9, 9E9, 9E9, 9E9, 9E9]];
	VAR jointtarget CDP_3396 := [[-8.19, 35.76, 6.02, 0, 48.22, -278.19], [9E9, 9E9, 9E9, 9E9, 9E9, 9E9]];
	VAR jointtarget CDP_3397 := [[-9.28, 35.94, 5.71, 0, 48.35, -279.28], [9E9, 9E9, 9E9, 9E9, 9E9, 9E9]];
	VAR jointtarget CDP_3398 := [[-10.36, 36.15, 5.36, 0, 48.5, -280.36], [9E9, 9E9, 9E9, 9E9, 9E9, 9E9]];
	VAR jointtarget CDP_3399 := [[-11.43, 36.37, 4.97, 0, 48.66, -281.43], [9E9, 9E9, 9E9, 9E9, 9E9, 9E9]];
	VAR jointtarget CDP_3400 := [[-11.44, 36.38, 4.96, 0, 48.66, -281.78], [9E9, 9E9, 9E9, 9E9, 9E9, 9E9]];
	VAR jointtarget CDP_3401 := [[-11.46, 36.38, 4.96, 0, 48.66, -282.45], [9E9, 9E9, 9E9, 9E9, 9E9, 9E9]];
	VAR jointtarget CDP_3402 := [[-11.48, 36.38, 4.95, 0, 48.67, -283.13], [9E9, 9E9, 9E9, 9E9, 9E9, 9E9]];
	VAR jointtarget CDP_3403 := [[-11.49, 36.39, 4.94, 0, 48.67, -283.81], [9E9, 9E9, 9E9, 9E9, 9E9, 9E9]];
	VAR jointtarget CDP_3404 := [[-11.51, 36.39, 4.93, 0, 48.67, -284.49], [9E9, 9E9, 9E9, 9E9, 9E9, 9E9]];
	VAR jointtarget CDP_3405 := [[-11.53, 36.4, 4.93, 0, 48.68, -285.17], [9E9, 9E9, 9E9, 9E9, 9E9, 9E9]];
	VAR jointtarget CDP_3406 := [[-11.54, 36.4, 4.92, 0, 48.68, -285.84], [9E9, 9E9, 9E9, 9E9, 9E9, 9E9]];
	VAR jointtarget CDP_3407 := [[-11.56, 36.41, 4.91, 0, 48.68, -286.52], [9E9, 9E9, 9E9, 9E9, 9E9, 9E9]];
	VAR jointtarget CDP_3408 := [[-11.57, 36.41, 4.9, 0, 48.69, -287.2], [9E9, 9E9, 9E9, 9E9, 9E9, 9E9]];
	VAR jointtarget CDP_3409 := [[-11.59, 36.42, 4.89, 0, 48.69, -287.88], [9E9, 9E9, 9E9, 9E9, 9E9, 9E9]];
	VAR jointtarget CDP_3410 := [[-11.6, 36.42, 4.88, 0, 48.7, -288.56], [9E9, 9E9, 9E9, 9E9, 9E9, 9E9]];
	VAR jointtarget CDP_3411 := [[-11.62, 36.43, 4.87, 0, 48.7, -289.23], [9E9, 9E9, 9E9, 9E9, 9E9, 9E9]];
	VAR jointtarget CDP_3412 := [[-11.64, 36.44, 4.86, 0, 48.71, -289.91], [9E9, 9E9, 9E9, 9E9, 9E9, 9E9]];
	VAR jointtarget CDP_3413 := [[-11.65, 36.44, 4.85, 0, 48.71, -290.59], [9E9, 9E9, 9E9, 9E9, 9E9, 9E9]];
	VAR jointtarget CDP_3414 := [[-11.67, 36.45, 4.84, 0, 48.72, -291.27], [9E9, 9E9, 9E9, 9E9, 9E9, 9E9]];
	VAR jointtarget CDP_3415 := [[-11.68, 36.46, 4.82, 0, 48.72, -291.94], [9E9, 9E9, 9E9, 9E9, 9E9, 9E9]];
	VAR jointtarget CDP_3416 := [[-11.7, 36.46, 4.81, 0, 48.73, -292.62], [9E9, 9E9, 9E9, 9E9, 9E9, 9E9]];
	VAR jointtarget CDP_3417 := [[-11.71, 36.47, 4.8, 0, 48.73, -293.3], [9E9, 9E9, 9E9, 9E9, 9E9, 9E9]];
	VAR jointtarget CDP_3418 := [[-11.73, 36.48, 4.79, 0, 48.74, -293.98], [9E9, 9E9, 9E9, 9E9, 9E9, 9E9]];
	VAR jointtarget CDP_3419 := [[-11.74, 36.49, 4.77, 0, 48.74, -294.65], [9E9, 9E9, 9E9, 9E9, 9E9, 9E9]];
	VAR jointtarget CDP_3420 := [[-11.8, 36.52, 4.72, 0, 48.76, -295.04], [9E9, 9E9, 9E9, 9E9, 9E9, 9E9]];
	VAR jointtarget CDP_3421 := [[-11.86, 36.55, 4.67, 0, 48.79, -295.11], [9E9, 9E9, 9E9, 9E9, 9E9, 9E9]];
	VAR jointtarget CDP_3422 := [[-11.93, 36.58, 4.61, 0, 48.81, -295.17], [9E9, 9E9, 9E9, 9E9, 9E9, 9E9]];
	VAR jointtarget CDP_3423 := [[-11.99, 36.61, 4.56, 0, 48.83, -295.23], [9E9, 9E9, 9E9, 9E9, 9E9, 9E9]];
	VAR jointtarget CDP_3424 := [[-12.05, 36.64, 4.5, 0, 48.85, -295.29], [9E9, 9E9, 9E9, 9E9, 9E9, 9E9]];
	VAR jointtarget CDP_3425 := [[-12.11, 36.67, 4.45, 0, 48.88, -295.35], [9E9, 9E9, 9E9, 9E9, 9E9, 9E9]];
	VAR jointtarget CDP_3426 := [[-12.17, 36.71, 4.4, 0, 48.9, -295.41], [9E9, 9E9, 9E9, 9E9, 9E9, 9E9]];
	VAR jointtarget CDP_3427 := [[-12.23, 36.74, 4.34, 0, 48.92, -295.47], [9E9, 9E9, 9E9, 9E9, 9E9, 9E9]];
	VAR jointtarget CDP_3428 := [[-12.29, 36.77, 4.29, 0, 48.94, -295.53], [9E9, 9E9, 9E9, 9E9, 9E9, 9E9]];
	VAR jointtarget CDP_3429 := [[-12.35, 36.8, 4.23, 0, 48.97, -295.59], [9E9, 9E9, 9E9, 9E9, 9E9, 9E9]];
	VAR jointtarget CDP_3430 := [[-12.41, 36.83, 4.18, 0, 48.99, -295.65], [9E9, 9E9, 9E9, 9E9, 9E9, 9E9]];
	VAR jointtarget CDP_3431 := [[-12.47, 36.87, 4.12, 0, 49.01, -295.71], [9E9, 9E9, 9E9, 9E9, 9E9, 9E9]];
	VAR jointtarget CDP_3432 := [[-12.53, 36.9, 4.07, 0, 49.04, -295.77], [9E9, 9E9, 9E9, 9E9, 9E9, 9E9]];
	VAR jointtarget CDP_3433 := [[-12.59, 36.93, 4.01, 0, 49.06, -295.83], [9E9, 9E9, 9E9, 9E9, 9E9, 9E9]];
	VAR jointtarget CDP_3434 := [[-12.65, 36.96, 3.95, 0, 49.08, -295.89], [9E9, 9E9, 9E9, 9E9, 9E9, 9E9]];
	VAR jointtarget CDP_3435 := [[-12.71, 36.99, 3.9, 0, 49.11, -295.95], [9E9, 9E9, 9E9, 9E9, 9E9, 9E9]];
	VAR jointtarget CDP_3436 := [[-12.77, 37.03, 3.84, 0, 49.13, -296.01], [9E9, 9E9, 9E9, 9E9, 9E9, 9E9]];
	VAR jointtarget CDP_3437 := [[-12.83, 37.06, 3.79, 0, 49.15, -296.07], [9E9, 9E9, 9E9, 9E9, 9E9, 9E9]];
	VAR jointtarget CDP_3438 := [[-12.89, 37.09, 3.73, 0, 49.18, -296.13], [9E9, 9E9, 9E9, 9E9, 9E9, 9E9]];
	VAR jointtarget CDP_3439 := [[-12.95, 37.12, 3.67, 0, 49.2, -296.19], [9E9, 9E9, 9E9, 9E9, 9E9, 9E9]];
	VAR jointtarget CDP_3440 := [[-13.07, 37.18, 3.58, 0, 49.24, -291.14], [9E9, 9E9, 9E9, 9E9, 9E9, 9E9]];
	VAR jointtarget CDP_3441 := [[-13.19, 37.2, 3.54, 0, 49.26, -280.95], [9E9, 9E9, 9E9, 9E9, 9E9, 9E9]];
	VAR jointtarget CDP_3442 := [[-13.32, 37.21, 3.53, 0, 49.26, -270.75], [9E9, 9E9, 9E9, 9E9, 9E9, 9E9]];
	VAR jointtarget CDP_3443 := [[-13.45, 37.18, 3.58, 0, 49.24, -260.55], [9E9, 9E9, 9E9, 9E9, 9E9, 9E9]];
	VAR jointtarget CDP_3444 := [[-13.57, 37.13, 3.66, 0, 49.21, -250.35], [9E9, 9E9, 9E9, 9E9, 9E9, 9E9]];
	VAR jointtarget CDP_3445 := [[-13.68, 37.06, 3.78, 0, 49.16, -240.14], [9E9, 9E9, 9E9, 9E9, 9E9, 9E9]];
	VAR jointtarget CDP_3446 := [[-13.78, 36.97, 3.94, 0, 49.09, -229.91], [9E9, 9E9, 9E9, 9E9, 9E9, 9E9]];
	VAR jointtarget CDP_3447 := [[-13.86, 36.86, 4.13, 0, 49.01, -219.67], [9E9, 9E9, 9E9, 9E9, 9E9, 9E9]];
	VAR jointtarget CDP_3448 := [[-13.93, 36.73, 4.35, 0, 48.92, -209.41], [9E9, 9E9, 9E9, 9E9, 9E9, 9E9]];
	VAR jointtarget CDP_3449 := [[-13.97, 36.6, 4.58, 0, 48.82, -199.13], [9E9, 9E9, 9E9, 9E9, 9E9, 9E9]];
	VAR jointtarget CDP_3450 := [[-13.99, 36.45, 4.83, 0, 48.72, -188.83], [9E9, 9E9, 9E9, 9E9, 9E9, 9E9]];
	VAR jointtarget CDP_3451 := [[-13.98, 36.31, 5.07, 0, 48.62, -178.5], [9E9, 9E9, 9E9, 9E9, 9E9, 9E9]];
	VAR jointtarget CDP_3452 := [[-13.96, 36.17, 5.31, 0, 48.52, -168.15], [9E9, 9E9, 9E9, 9E9, 9E9, 9E9]];
	VAR jointtarget CDP_3453 := [[-13.91, 36.04, 5.54, 0, 48.42, -157.77], [9E9, 9E9, 9E9, 9E9, 9E9, 9E9]];
	VAR jointtarget CDP_3454 := [[-13.84, 35.92, 5.75, 0, 48.34, -147.38], [9E9, 9E9, 9E9, 9E9, 9E9, 9E9]];
	VAR jointtarget CDP_3455 := [[-13.75, 35.81, 5.93, 0, 48.26, -136.97], [9E9, 9E9, 9E9, 9E9, 9E9, 9E9]];
	VAR jointtarget CDP_3456 := [[-13.64, 35.73, 6.07, 0, 48.2, -126.54], [9E9, 9E9, 9E9, 9E9, 9E9, 9E9]];
	VAR jointtarget CDP_3457 := [[-13.52, 35.67, 6.18, 0, 48.16, -116.09], [9E9, 9E9, 9E9, 9E9, 9E9, 9E9]];
	VAR jointtarget CDP_3458 := [[-13.4, 35.63, 6.24, 0, 48.13, -105.64], [9E9, 9E9, 9E9, 9E9, 9E9, 9E9]];
	VAR jointtarget CDP_3459 := [[-13.27, 35.61, 6.27, 0, 48.12, -95.19], [9E9, 9E9, 9E9, 9E9, 9E9, 9E9]];
	VAR jointtarget CDP_3460 := [[-13.2, 35.61, 6.27, 0, 48.12, -89.96], [9E9, 9E9, 9E9, 9E9, 9E9, 9E9]];
	VAR jointtarget CDP_3461 := [[-13.13, 35.61, 6.27, 0, 48.12, -89.89], [9E9, 9E9, 9E9, 9E9, 9E9, 9E9]];
	VAR jointtarget CDP_3462 := [[-13.06, 35.61, 6.27, 0, 48.12, -89.82], [9E9, 9E9, 9E9, 9E9, 9E9, 9E9]];
	VAR jointtarget CDP_3463 := [[-12.99, 35.61, 6.26, 0, 48.12, -89.75], [9E9, 9E9, 9E9, 9E9, 9E9, 9E9]];
	VAR jointtarget CDP_3464 := [[-12.93, 35.61, 6.26, 0, 48.12, -89.69], [9E9, 9E9, 9E9, 9E9, 9E9, 9E9]];
	VAR jointtarget CDP_3465 := [[-12.86, 35.61, 6.26, 0, 48.12, -89.62], [9E9, 9E9, 9E9, 9E9, 9E9, 9E9]];
	VAR jointtarget CDP_3466 := [[-12.79, 35.61, 6.26, 0, 48.13, -89.55], [9E9, 9E9, 9E9, 9E9, 9E9, 9E9]];
	VAR jointtarget CDP_3467 := [[-12.72, 35.61, 6.26, 0, 48.13, -89.48], [9E9, 9E9, 9E9, 9E9, 9E9, 9E9]];
	VAR jointtarget CDP_3468 := [[-12.65, 35.61, 6.26, 0, 48.13, -89.41], [9E9, 9E9, 9E9, 9E9, 9E9, 9E9]];
	VAR jointtarget CDP_3469 := [[-12.59, 35.61, 6.26, 0, 48.13, -89.35], [9E9, 9E9, 9E9, 9E9, 9E9, 9E9]];
	VAR jointtarget CDP_3470 := [[-12.52, 35.61, 6.26, 0, 48.13, -89.28], [9E9, 9E9, 9E9, 9E9, 9E9, 9E9]];
	VAR jointtarget CDP_3471 := [[-12.45, 35.61, 6.25, 0, 48.13, -89.21], [9E9, 9E9, 9E9, 9E9, 9E9, 9E9]];
	VAR jointtarget CDP_3472 := [[-12.38, 35.61, 6.25, 0, 48.13, -89.14], [9E9, 9E9, 9E9, 9E9, 9E9, 9E9]];
	VAR jointtarget CDP_3473 := [[-12.32, 35.61, 6.25, 0, 48.14, -89.07], [9E9, 9E9, 9E9, 9E9, 9E9, 9E9]];
	VAR jointtarget CDP_3474 := [[-12.25, 35.61, 6.25, 0, 48.14, -89.01], [9E9, 9E9, 9E9, 9E9, 9E9, 9E9]];
	VAR jointtarget CDP_3475 := [[-12.18, 35.62, 6.25, 0, 48.14, -88.94], [9E9, 9E9, 9E9, 9E9, 9E9, 9E9]];
	VAR jointtarget CDP_3476 := [[-12.11, 35.62, 6.24, 0, 48.14, -88.87], [9E9, 9E9, 9E9, 9E9, 9E9, 9E9]];
	VAR jointtarget CDP_3477 := [[-12.04, 35.62, 6.24, 0, 48.14, -88.8], [9E9, 9E9, 9E9, 9E9, 9E9, 9E9]];
	VAR jointtarget CDP_3478 := [[-11.98, 35.62, 6.24, 0, 48.14, -88.74], [9E9, 9E9, 9E9, 9E9, 9E9, 9E9]];
	VAR jointtarget CDP_3479 := [[-11.91, 35.62, 6.24, 0, 48.15, -88.67], [9E9, 9E9, 9E9, 9E9, 9E9, 9E9]];
	VAR jointtarget CDP_3480 := [[-11.89, 35.62, 6.23, 0, 48.15, -88.98], [9E9, 9E9, 9E9, 9E9, 9E9, 9E9]];
	VAR jointtarget CDP_3481 := [[-11.87, 35.62, 6.23, 0, 48.15, -89.63], [9E9, 9E9, 9E9, 9E9, 9E9, 9E9]];
	VAR jointtarget CDP_3482 := [[-11.86, 35.62, 6.23, 0, 48.15, -90.27], [9E9, 9E9, 9E9, 9E9, 9E9, 9E9]];
	VAR jointtarget CDP_3483 := [[-11.84, 35.62, 6.24, 0, 48.15, -90.92], [9E9, 9E9, 9E9, 9E9, 9E9, 9E9]];
	VAR jointtarget CDP_3484 := [[-11.82, 35.62, 6.24, 0, 48.15, -91.56], [9E9, 9E9, 9E9, 9E9, 9E9, 9E9]];
	VAR jointtarget CDP_3485 := [[-11.81, 35.62, 6.24, 0, 48.15, -92.21], [9E9, 9E9, 9E9, 9E9, 9E9, 9E9]];
	VAR jointtarget CDP_3486 := [[-11.79, 35.62, 6.24, 0, 48.14, -92.85], [9E9, 9E9, 9E9, 9E9, 9E9, 9E9]];
	VAR jointtarget CDP_3487 := [[-11.77, 35.62, 6.24, 0, 48.14, -93.5], [9E9, 9E9, 9E9, 9E9, 9E9, 9E9]];
	VAR jointtarget CDP_3488 := [[-11.76, 35.61, 6.24, 0, 48.14, -94.14], [9E9, 9E9, 9E9, 9E9, 9E9, 9E9]];
	VAR jointtarget CDP_3489 := [[-11.74, 35.61, 6.25, 0, 48.14, -94.79], [9E9, 9E9, 9E9, 9E9, 9E9, 9E9]];
	VAR jointtarget CDP_3490 := [[-11.72, 35.61, 6.25, 0, 48.14, -95.43], [9E9, 9E9, 9E9, 9E9, 9E9, 9E9]];
	VAR jointtarget CDP_3491 := [[-11.71, 35.61, 6.25, 0, 48.14, -96.08], [9E9, 9E9, 9E9, 9E9, 9E9, 9E9]];
	VAR jointtarget CDP_3492 := [[-11.69, 35.61, 6.26, 0, 48.14, -96.72], [9E9, 9E9, 9E9, 9E9, 9E9, 9E9]];
	VAR jointtarget CDP_3493 := [[-11.67, 35.6, 6.26, 0, 48.14, -97.37], [9E9, 9E9, 9E9, 9E9, 9E9, 9E9]];
	VAR jointtarget CDP_3494 := [[-11.66, 35.6, 6.26, 0, 48.14, -98.01], [9E9, 9E9, 9E9, 9E9, 9E9, 9E9]];
	VAR jointtarget CDP_3495 := [[-11.64, 35.6, 6.27, 0, 48.13, -98.66], [9E9, 9E9, 9E9, 9E9, 9E9, 9E9]];
	VAR jointtarget CDP_3496 := [[-11.62, 35.6, 6.27, 0, 48.13, -99.31], [9E9, 9E9, 9E9, 9E9, 9E9, 9E9]];
	VAR jointtarget CDP_3497 := [[-11.61, 35.59, 6.28, 0, 48.13, -99.95], [9E9, 9E9, 9E9, 9E9, 9E9, 9E9]];
	VAR jointtarget CDP_3498 := [[-11.59, 35.59, 6.28, 0, 48.13, -100.6], [9E9, 9E9, 9E9, 9E9, 9E9, 9E9]];
	VAR jointtarget CDP_3499 := [[-11.57, 35.59, 6.29, 0, 48.12, -101.24], [9E9, 9E9, 9E9, 9E9, 9E9, 9E9]];
	VAR jointtarget CDP_3500 := [[-10.48, 35.36, 6.68, 0, 47.96, -100.48], [9E9, 9E9, 9E9, 9E9, 9E9, 9E9]];
	VAR jointtarget CDP_3501 := [[-9.38, 35.15, 7.03, 0, 47.82, -99.38], [9E9, 9E9, 9E9, 9E9, 9E9, 9E9]];
	VAR jointtarget CDP_3502 := [[-8.27, 34.97, 7.35, 0, 47.69, -98.27], [9E9, 9E9, 9E9, 9E9, 9E9, 9E9]];
	VAR jointtarget CDP_3503 := [[-7.15, 34.81, 7.62, 0, 47.58, -97.15], [9E9, 9E9, 9E9, 9E9, 9E9, 9E9]];
	VAR jointtarget CDP_3504 := [[-6.03, 34.67, 7.85, 0, 47.48, -96.03], [9E9, 9E9, 9E9, 9E9, 9E9, 9E9]];
	VAR jointtarget CDP_3505 := [[-4.9, 34.56, 8.04, 0, 47.4, -94.9], [9E9, 9E9, 9E9, 9E9, 9E9, 9E9]];
	VAR jointtarget CDP_3506 := [[-3.77, 34.47, 8.2, 0, 47.34, -93.77], [9E9, 9E9, 9E9, 9E9, 9E9, 9E9]];
	VAR jointtarget CDP_3507 := [[-2.64, 34.4, 8.31, 0, 47.29, -92.64], [9E9, 9E9, 9E9, 9E9, 9E9, 9E9]];
	VAR jointtarget CDP_3508 := [[-1.51, 34.36, 8.38, 0, 47.26, -91.51], [9E9, 9E9, 9E9, 9E9, 9E9, 9E9]];
	VAR jointtarget CDP_3509 := [[-0.37, 34.34, 8.42, 0, 47.25, -90.37], [9E9, 9E9, 9E9, 9E9, 9E9, 9E9]];
	VAR jointtarget CDP_3510 := [[0.76, 34.34, 8.41, 0, 47.25, -89.24], [9E9, 9E9, 9E9, 9E9, 9E9, 9E9]];
	VAR jointtarget CDP_3511 := [[1.9, 34.37, 8.36, 0, 47.27, -88.1], [9E9, 9E9, 9E9, 9E9, 9E9, 9E9]];
	VAR jointtarget CDP_3512 := [[3.03, 34.42, 8.28, 0, 47.3, -86.97], [9E9, 9E9, 9E9, 9E9, 9E9, 9E9]];
	VAR jointtarget CDP_3513 := [[4.16, 34.49, 8.15, 0, 47.36, -85.84], [9E9, 9E9, 9E9, 9E9, 9E9, 9E9]];
	VAR jointtarget CDP_3514 := [[5.29, 34.59, 7.98, 0, 47.43, -84.71], [9E9, 9E9, 9E9, 9E9, 9E9, 9E9]];
	VAR jointtarget CDP_3515 := [[6.42, 34.71, 7.78, 0, 47.51, -83.58], [9E9, 9E9, 9E9, 9E9, 9E9, 9E9]];
	VAR jointtarget CDP_3516 := [[7.54, 34.86, 7.53, 0, 47.61, -82.46], [9E9, 9E9, 9E9, 9E9, 9E9, 9E9]];
	VAR jointtarget CDP_3517 := [[8.65, 35.03, 7.24, 0, 47.73, -81.35], [9E9, 9E9, 9E9, 9E9, 9E9, 9E9]];
	VAR jointtarget CDP_3518 := [[9.76, 35.22, 6.92, 0, 47.86, -80.24], [9E9, 9E9, 9E9, 9E9, 9E9, 9E9]];
	VAR jointtarget CDP_3519 := [[10.86, 35.43, 6.55, 0, 48.02, -79.14], [9E9, 9E9, 9E9, 9E9, 9E9, 9E9]];
	VAR jointtarget CDP_3520 := [[10.87, 35.44, 6.55, 0, 48.02, -79.46], [9E9, 9E9, 9E9, 9E9, 9E9, 9E9]];
	VAR jointtarget CDP_3521 := [[10.89, 35.44, 6.54, 0, 48.02, -80.1], [9E9, 9E9, 9E9, 9E9, 9E9, 9E9]];
	VAR jointtarget CDP_3522 := [[10.91, 35.44, 6.54, 0, 48.02, -80.75], [9E9, 9E9, 9E9, 9E9, 9E9, 9E9]];
	VAR jointtarget CDP_3523 := [[10.92, 35.44, 6.53, 0, 48.02, -81.39], [9E9, 9E9, 9E9, 9E9, 9E9, 9E9]];
	VAR jointtarget CDP_3524 := [[10.94, 35.45, 6.53, 0, 48.03, -82.04], [9E9, 9E9, 9E9, 9E9, 9E9, 9E9]];
	VAR jointtarget CDP_3525 := [[10.96, 35.45, 6.52, 0, 48.03, -82.68], [9E9, 9E9, 9E9, 9E9, 9E9, 9E9]];
	VAR jointtarget CDP_3526 := [[10.97, 35.45, 6.52, 0, 48.03, -83.33], [9E9, 9E9, 9E9, 9E9, 9E9, 9E9]];
	VAR jointtarget CDP_3527 := [[10.99, 35.45, 6.52, 0, 48.03, -83.97], [9E9, 9E9, 9E9, 9E9, 9E9, 9E9]];
	VAR jointtarget CDP_3528 := [[11.01, 35.46, 6.51, 0, 48.03, -84.62], [9E9, 9E9, 9E9, 9E9, 9E9, 9E9]];
	VAR jointtarget CDP_3529 := [[11.02, 35.46, 6.51, 0, 48.03, -85.27], [9E9, 9E9, 9E9, 9E9, 9E9, 9E9]];
	VAR jointtarget CDP_3530 := [[11.04, 35.46, 6.51, 0, 48.03, -85.91], [9E9, 9E9, 9E9, 9E9, 9E9, 9E9]];
	VAR jointtarget CDP_3531 := [[11.06, 35.46, 6.51, 0, 48.03, -86.56], [9E9, 9E9, 9E9, 9E9, 9E9, 9E9]];
	VAR jointtarget CDP_3532 := [[11.07, 35.46, 6.5, 0, 48.04, -87.2], [9E9, 9E9, 9E9, 9E9, 9E9, 9E9]];
	VAR jointtarget CDP_3533 := [[11.09, 35.46, 6.5, 0, 48.04, -87.85], [9E9, 9E9, 9E9, 9E9, 9E9, 9E9]];
	VAR jointtarget CDP_3534 := [[11.11, 35.46, 6.5, 0, 48.04, -88.49], [9E9, 9E9, 9E9, 9E9, 9E9, 9E9]];
	VAR jointtarget CDP_3535 := [[11.13, 35.46, 6.5, 0, 48.04, -89.14], [9E9, 9E9, 9E9, 9E9, 9E9, 9E9]];
	VAR jointtarget CDP_3536 := [[11.14, 35.46, 6.5, 0, 48.04, -89.78], [9E9, 9E9, 9E9, 9E9, 9E9, 9E9]];
	VAR jointtarget CDP_3537 := [[11.16, 35.46, 6.5, 0, 48.04, -90.43], [9E9, 9E9, 9E9, 9E9, 9E9, 9E9]];
	VAR jointtarget CDP_3538 := [[11.18, 35.46, 6.5, 0, 48.04, -91.07], [9E9, 9E9, 9E9, 9E9, 9E9, 9E9]];
	VAR jointtarget CDP_3539 := [[11.19, 35.46, 6.5, 0, 48.04, -91.72], [9E9, 9E9, 9E9, 9E9, 9E9, 9E9]];
	VAR jointtarget CDP_3540 := [[11.26, 35.46, 6.51, 0, 48.03, -91.98], [9E9, 9E9, 9E9, 9E9, 9E9, 9E9]];
	VAR jointtarget CDP_3541 := [[11.33, 35.46, 6.51, 0, 48.03, -91.91], [9E9, 9E9, 9E9, 9E9, 9E9, 9E9]];
	VAR jointtarget CDP_3542 := [[11.4, 35.45, 6.52, 0, 48.03, -91.84], [9E9, 9E9, 9E9, 9E9, 9E9, 9E9]];
	VAR jointtarget CDP_3543 := [[11.47, 35.45, 6.52, 0, 48.03, -91.78], [9E9, 9E9, 9E9, 9E9, 9E9, 9E9]];
	VAR jointtarget CDP_3544 := [[11.53, 35.45, 6.52, 0, 48.03, -91.71], [9E9, 9E9, 9E9, 9E9, 9E9, 9E9]];
	VAR jointtarget CDP_3545 := [[11.6, 35.45, 6.53, 0, 48.03, -91.64], [9E9, 9E9, 9E9, 9E9, 9E9, 9E9]];
	VAR jointtarget CDP_3546 := [[11.67, 35.44, 6.53, 0, 48.02, -91.57], [9E9, 9E9, 9E9, 9E9, 9E9, 9E9]];
	VAR jointtarget CDP_3547 := [[11.74, 35.44, 6.53, 0, 48.02, -91.5], [9E9, 9E9, 9E9, 9E9, 9E9, 9E9]];
	VAR jointtarget CDP_3548 := [[11.81, 35.44, 6.54, 0, 48.02, -91.44], [9E9, 9E9, 9E9, 9E9, 9E9, 9E9]];
	VAR jointtarget CDP_3549 := [[11.87, 35.44, 6.54, 0, 48.02, -91.37], [9E9, 9E9, 9E9, 9E9, 9E9, 9E9]];
	VAR jointtarget CDP_3550 := [[11.94, 35.44, 6.54, 0, 48.02, -91.3], [9E9, 9E9, 9E9, 9E9, 9E9, 9E9]];
	VAR jointtarget CDP_3551 := [[12.01, 35.44, 6.55, 0, 48.02, -91.23], [9E9, 9E9, 9E9, 9E9, 9E9, 9E9]];
	VAR jointtarget CDP_3552 := [[12.08, 35.43, 6.55, 0, 48.02, -91.16], [9E9, 9E9, 9E9, 9E9, 9E9, 9E9]];
	VAR jointtarget CDP_3553 := [[12.15, 35.43, 6.55, 0, 48.02, -91.09], [9E9, 9E9, 9E9, 9E9, 9E9, 9E9]];
	VAR jointtarget CDP_3554 := [[12.21, 35.43, 6.55, 0, 48.01, -91.03], [9E9, 9E9, 9E9, 9E9, 9E9, 9E9]];
	VAR jointtarget CDP_3555 := [[12.28, 35.43, 6.56, 0, 48.01, -90.96], [9E9, 9E9, 9E9, 9E9, 9E9, 9E9]];
	VAR jointtarget CDP_3556 := [[12.35, 35.43, 6.56, 0, 48.01, -90.89], [9E9, 9E9, 9E9, 9E9, 9E9, 9E9]];
	VAR jointtarget CDP_3557 := [[12.42, 35.43, 6.56, 0, 48.01, -90.82], [9E9, 9E9, 9E9, 9E9, 9E9, 9E9]];
	VAR jointtarget CDP_3558 := [[12.49, 35.43, 6.56, 0, 48.01, -90.75], [9E9, 9E9, 9E9, 9E9, 9E9, 9E9]];
	VAR jointtarget CDP_3559 := [[12.55, 35.43, 6.56, 0, 48.01, -90.69], [9E9, 9E9, 9E9, 9E9, 9E9, 9E9]];
	VAR jointtarget CDP_3560 := [[12.69, 35.44, 6.54, 0, 48.02, -85.39], [9E9, 9E9, 9E9, 9E9, 9E9, 9E9]];
	VAR jointtarget CDP_3561 := [[12.81, 35.47, 6.48, 0, 48.04, -74.94], [9E9, 9E9, 9E9, 9E9, 9E9, 9E9]];
	VAR jointtarget CDP_3562 := [[12.93, 35.53, 6.38, 0, 48.09, -64.5], [9E9, 9E9, 9E9, 9E9, 9E9, 9E9]];
	VAR jointtarget CDP_3563 := [[13.04, 35.62, 6.23, 0, 48.15, -54.07], [9E9, 9E9, 9E9, 9E9, 9E9, 9E9]];
	VAR jointtarget CDP_3564 := [[13.13, 35.72, 6.06, 0, 48.22, -43.65], [9E9, 9E9, 9E9, 9E9, 9E9, 9E9]];
	VAR jointtarget CDP_3565 := [[13.2, 35.84, 5.85, 0, 48.31, -33.25], [9E9, 9E9, 9E9, 9E9, 9E9, 9E9]];
	VAR jointtarget CDP_3566 := [[13.25, 35.97, 5.63, 0, 48.4, -22.88], [9E9, 9E9, 9E9, 9E9, 9E9, 9E9]];
	VAR jointtarget CDP_3567 := [[13.28, 36.11, 5.39, 0, 48.5, -12.53], [9E9, 9E9, 9E9, 9E9, 9E9, 9E9]];
	VAR jointtarget CDP_3568 := [[13.29, 36.25, 5.14, 0, 48.6, -2.2], [9E9, 9E9, 9E9, 9E9, 9E9, 9E9]];
	VAR jointtarget CDP_3569 := [[13.27, 36.4, 4.9, 0, 48.7, 8.11], [9E9, 9E9, 9E9, 9E9, 9E9, 9E9]];
	VAR jointtarget CDP_3570 := [[13.23, 36.53, 4.67, 0, 48.8, 18.39], [9E9, 9E9, 9E9, 9E9, 9E9, 9E9]];
	VAR jointtarget CDP_3571 := [[13.17, 36.66, 4.45, 0, 48.89, 28.65], [9E9, 9E9, 9E9, 9E9, 9E9, 9E9]];
	VAR jointtarget CDP_3572 := [[13.08, 36.77, 4.26, 0, 48.97, 38.9], [9E9, 9E9, 9E9, 9E9, 9E9, 9E9]];
	VAR jointtarget CDP_3573 := [[12.99, 36.87, 4.1, 0, 49.04, 49.12], [9E9, 9E9, 9E9, 9E9, 9E9, 9E9]];
	VAR jointtarget CDP_3574 := [[12.88, 36.94, 3.97, 0, 49.09, 59.33], [9E9, 9E9, 9E9, 9E9, 9E9, 9E9]];
	VAR jointtarget CDP_3575 := [[12.75, 36.99, 3.88, 0, 49.13, 69.54], [9E9, 9E9, 9E9, 9E9, 9E9, 9E9]];
	VAR jointtarget CDP_3576 := [[12.63, 37.01, 3.84, 0, 49.15, 79.73], [9E9, 9E9, 9E9, 9E9, 9E9, 9E9]];
	VAR jointtarget CDP_3577 := [[12.5, 37.01, 3.84, 0, 49.15, 89.93], [9E9, 9E9, 9E9, 9E9, 9E9, 9E9]];
	VAR jointtarget CDP_3578 := [[12.37, 36.99, 3.88, 0, 49.13, 100.13], [9E9, 9E9, 9E9, 9E9, 9E9, 9E9]];
	VAR jointtarget CDP_3579 := [[12.25, 36.94, 3.97, 0, 49.09, 110.33], [9E9, 9E9, 9E9, 9E9, 9E9, 9E9]];
	VAR jointtarget CDP_3580 := [[12.19, 36.91, 4.02, 0, 49.07, 115.43], [9E9, 9E9, 9E9, 9E9, 9E9, 9E9]];
	VAR jointtarget CDP_3581 := [[12.13, 36.87, 4.08, 0, 49.05, 115.37], [9E9, 9E9, 9E9, 9E9, 9E9, 9E9]];
	VAR jointtarget CDP_3582 := [[12.07, 36.84, 4.13, 0, 49.02, 115.31], [9E9, 9E9, 9E9, 9E9, 9E9, 9E9]];
	VAR jointtarget CDP_3583 := [[12.01, 36.81, 4.19, 0, 49, 115.25], [9E9, 9E9, 9E9, 9E9, 9E9, 9E9]];
	VAR jointtarget CDP_3584 := [[11.95, 36.78, 4.24, 0, 48.98, 115.19], [9E9, 9E9, 9E9, 9E9, 9E9, 9E9]];
	VAR jointtarget CDP_3585 := [[11.89, 36.75, 4.3, 0, 48.95, 115.13], [9E9, 9E9, 9E9, 9E9, 9E9, 9E9]];
	VAR jointtarget CDP_3586 := [[11.83, 36.72, 4.35, 0, 48.93, 115.07], [9E9, 9E9, 9E9, 9E9, 9E9, 9E9]];
	VAR jointtarget CDP_3587 := [[11.77, 36.69, 4.4, 0, 48.91, 115.01], [9E9, 9E9, 9E9, 9E9, 9E9, 9E9]];
	VAR jointtarget CDP_3588 := [[11.71, 36.65, 4.46, 0, 48.89, 114.95], [9E9, 9E9, 9E9, 9E9, 9E9, 9E9]];
	VAR jointtarget CDP_3589 := [[11.65, 36.62, 4.51, 0, 48.86, 114.89], [9E9, 9E9, 9E9, 9E9, 9E9, 9E9]];
	VAR jointtarget CDP_3590 := [[11.59, 36.59, 4.57, 0, 48.84, 114.83], [9E9, 9E9, 9E9, 9E9, 9E9, 9E9]];
	VAR jointtarget CDP_3591 := [[11.53, 36.56, 4.62, 0, 48.82, 114.77], [9E9, 9E9, 9E9, 9E9, 9E9, 9E9]];
	VAR jointtarget CDP_3592 := [[11.47, 36.53, 4.67, 0, 48.8, 114.71], [9E9, 9E9, 9E9, 9E9, 9E9, 9E9]];
	VAR jointtarget CDP_3593 := [[11.4, 36.5, 4.72, 0, 48.78, 114.64], [9E9, 9E9, 9E9, 9E9, 9E9, 9E9]];
	VAR jointtarget CDP_3594 := [[11.34, 36.47, 4.78, 0, 48.75, 114.58], [9E9, 9E9, 9E9, 9E9, 9E9, 9E9]];
	VAR jointtarget CDP_3595 := [[11.28, 36.44, 4.83, 0, 48.73, 114.52], [9E9, 9E9, 9E9, 9E9, 9E9, 9E9]];
	VAR jointtarget CDP_3596 := [[11.22, 36.41, 4.88, 0, 48.71, 114.46], [9E9, 9E9, 9E9, 9E9, 9E9, 9E9]];
	VAR jointtarget CDP_3597 := [[11.16, 36.38, 4.94, 0, 48.69, 114.4], [9E9, 9E9, 9E9, 9E9, 9E9, 9E9]];
	VAR jointtarget CDP_3598 := [[11.1, 36.35, 4.99, 0, 48.67, 114.34], [9E9, 9E9, 9E9, 9E9, 9E9, 9E9]];
	VAR jointtarget CDP_3599 := [[11.04, 36.32, 5.04, 0, 48.64, 114.28], [9E9, 9E9, 9E9, 9E9, 9E9, 9E9]];
	VAR jointtarget CDP_3600 := [[11.02, 36.31, 5.05, 0, 48.64, 113.93], [9E9, 9E9, 9E9, 9E9, 9E9, 9E9]];
	VAR jointtarget CDP_3601 := [[11.01, 36.3, 5.06, 0, 48.63, 113.26], [9E9, 9E9, 9E9, 9E9, 9E9, 9E9]];
	VAR jointtarget CDP_3602 := [[10.99, 36.29, 5.08, 0, 48.63, 112.58], [9E9, 9E9, 9E9, 9E9, 9E9, 9E9]];
	VAR jointtarget CDP_3603 := [[10.98, 36.29, 5.09, 0, 48.62, 111.9], [9E9, 9E9, 9E9, 9E9, 9E9, 9E9]];
	VAR jointtarget CDP_3604 := [[10.96, 36.28, 5.1, 0, 48.62, 111.22], [9E9, 9E9, 9E9, 9E9, 9E9, 9E9]];
	VAR jointtarget CDP_3605 := [[10.95, 36.27, 5.11, 0, 48.61, 110.55], [9E9, 9E9, 9E9, 9E9, 9E9, 9E9]];
	VAR jointtarget CDP_3606 := [[10.93, 36.27, 5.12, 0, 48.61, 109.87], [9E9, 9E9, 9E9, 9E9, 9E9, 9E9]];
	VAR jointtarget CDP_3607 := [[10.91, 36.26, 5.13, 0, 48.61, 109.19], [9E9, 9E9, 9E9, 9E9, 9E9, 9E9]];
	VAR jointtarget CDP_3608 := [[10.9, 36.26, 5.14, 0, 48.6, 108.51], [9E9, 9E9, 9E9, 9E9, 9E9, 9E9]];
	VAR jointtarget CDP_3609 := [[10.88, 36.25, 5.15, 0, 48.6, 107.83], [9E9, 9E9, 9E9, 9E9, 9E9, 9E9]];
	VAR jointtarget CDP_3610 := [[10.87, 36.25, 5.16, 0, 48.59, 107.16], [9E9, 9E9, 9E9, 9E9, 9E9, 9E9]];
	VAR jointtarget CDP_3611 := [[10.85, 36.24, 5.17, 0, 48.59, 106.48], [9E9, 9E9, 9E9, 9E9, 9E9, 9E9]];
	VAR jointtarget CDP_3612 := [[10.83, 36.24, 5.18, 0, 48.59, 105.8], [9E9, 9E9, 9E9, 9E9, 9E9, 9E9]];
	VAR jointtarget CDP_3613 := [[10.82, 36.23, 5.19, 0, 48.58, 105.12], [9E9, 9E9, 9E9, 9E9, 9E9, 9E9]];
	VAR jointtarget CDP_3614 := [[10.8, 36.23, 5.19, 0, 48.58, 104.44], [9E9, 9E9, 9E9, 9E9, 9E9, 9E9]];
	VAR jointtarget CDP_3615 := [[10.79, 36.22, 5.2, 0, 48.58, 103.77], [9E9, 9E9, 9E9, 9E9, 9E9, 9E9]];
	VAR jointtarget CDP_3616 := [[10.77, 36.22, 5.21, 0, 48.57, 103.09], [9E9, 9E9, 9E9, 9E9, 9E9, 9E9]];
	VAR jointtarget CDP_3617 := [[10.75, 36.21, 5.22, 0, 48.57, 102.41], [9E9, 9E9, 9E9, 9E9, 9E9, 9E9]];
	VAR jointtarget CDP_3618 := [[10.74, 36.21, 5.22, 0, 48.57, 101.73], [9E9, 9E9, 9E9, 9E9, 9E9, 9E9]];
	VAR jointtarget CDP_3619 := [[10.72, 36.21, 5.23, 0, 48.57, 101.05], [9E9, 9E9, 9E9, 9E9, 9E9, 9E9]];
	VAR jointtarget CDP_3620 := [[9.64, 36, 5.59, 0, 48.42, 99.64], [9E9, 9E9, 9E9, 9E9, 9E9, 9E9]];
	VAR jointtarget CDP_3621 := [[8.56, 35.81, 5.91, 0, 48.28, 98.56], [9E9, 9E9, 9E9, 9E9, 9E9, 9E9]];
	VAR jointtarget CDP_3622 := [[7.47, 35.64, 6.2, 0, 48.16, 97.47], [9E9, 9E9, 9E9, 9E9, 9E9, 9E9]];
	VAR jointtarget CDP_3623 := [[6.38, 35.5, 6.44, 0, 48.06, 96.38], [9E9, 9E9, 9E9, 9E9, 9E9, 9E9]];
	VAR jointtarget CDP_3624 := [[5.28, 35.38, 6.65, 0, 47.98, 95.28], [9E9, 9E9, 9E9, 9E9, 9E9, 9E9]];
	VAR jointtarget CDP_3625 := [[4.17, 35.28, 6.81, 0, 47.91, 94.17], [9E9, 9E9, 9E9, 9E9, 9E9, 9E9]];
	VAR jointtarget CDP_3626 := [[3.07, 35.2, 6.94, 0, 47.85, 93.07], [9E9, 9E9, 9E9, 9E9, 9E9, 9E9]];
	VAR jointtarget CDP_3627 := [[1.96, 35.15, 7.03, 0, 47.82, 91.96], [9E9, 9E9, 9E9, 9E9, 9E9, 9E9]];
	VAR jointtarget CDP_3628 := [[0.85, 35.12, 7.08, 0, 47.8, 90.85], [9E9, 9E9, 9E9, 9E9, 9E9, 9E9]];
	VAR jointtarget CDP_3629 := [[-0.26, 35.12, 7.09, 0, 47.79, 89.74], [9E9, 9E9, 9E9, 9E9, 9E9, 9E9]];
	VAR jointtarget CDP_3630 := [[-1.37, 35.13, 7.06, 0, 47.81, 88.63], [9E9, 9E9, 9E9, 9E9, 9E9, 9E9]];
	VAR jointtarget CDP_3631 := [[-2.48, 35.17, 6.99, 0, 47.83, 87.52], [9E9, 9E9, 9E9, 9E9, 9E9, 9E9]];
	VAR jointtarget CDP_3632 := [[-3.59, 35.24, 6.89, 0, 47.88, 86.41], [9E9, 9E9, 9E9, 9E9, 9E9, 9E9]];
	VAR jointtarget CDP_3633 := [[-4.7, 35.32, 6.74, 0, 47.94, 85.3], [9E9, 9E9, 9E9, 9E9, 9E9, 9E9]];
	VAR jointtarget CDP_3634 := [[-5.8, 35.43, 6.55, 0, 48.01, 84.2], [9E9, 9E9, 9E9, 9E9, 9E9, 9E9]];
	VAR jointtarget CDP_3635 := [[-6.9, 35.56, 6.33, 0, 48.11, 83.1], [9E9, 9E9, 9E9, 9E9, 9E9, 9E9]];
	VAR jointtarget CDP_3636 := [[-7.99, 35.72, 6.07, 0, 48.22, 82.01], [9E9, 9E9, 9E9, 9E9, 9E9, 9E9]];
	VAR jointtarget CDP_3637 := [[-9.08, 35.89, 5.76, 0, 48.34, 80.92], [9E9, 9E9, 9E9, 9E9, 9E9, 9E9]];
	VAR jointtarget CDP_3638 := [[-10.16, 36.09, 5.42, 0, 48.48, 79.84], [9E9, 9E9, 9E9, 9E9, 9E9, 9E9]];
	VAR jointtarget CDP_3639 := [[-11.23, 36.31, 5.04, 0, 48.64, 78.77], [9E9, 9E9, 9E9, 9E9, 9E9, 9E9]];
	VAR jointtarget CDP_3640 := [[-11.28, 36.33, 5.02, 0, 48.65, 79.81], [9E9, 9E9, 9E9, 9E9, 9E9, 9E9]];
	VAR jointtarget CDP_3641 := [[-11.34, 36.33, 5.01, 0, 48.66, 81.95], [9E9, 9E9, 9E9, 9E9, 9E9, 9E9]];
	VAR jointtarget CDP_3642 := [[-11.39, 36.34, 5, 0, 48.66, 84.09], [9E9, 9E9, 9E9, 9E9, 9E9, 9E9]];
	VAR jointtarget CDP_3643 := [[-11.45, 36.34, 4.99, 0, 48.66, 86.23], [9E9, 9E9, 9E9, 9E9, 9E9, 9E9]];
	VAR jointtarget CDP_3644 := [[-11.5, 36.35, 4.99, 0, 48.67, 88.37], [9E9, 9E9, 9E9, 9E9, 9E9, 9E9]];
	VAR jointtarget CDP_3645 := [[-11.56, 36.35, 4.99, 0, 48.67, 90.51], [9E9, 9E9, 9E9, 9E9, 9E9, 9E9]];
	VAR jointtarget CDP_3646 := [[-11.61, 36.34, 4.99, 0, 48.66, 92.65], [9E9, 9E9, 9E9, 9E9, 9E9, 9E9]];
	VAR jointtarget CDP_3647 := [[-11.67, 36.34, 5, 0, 48.66, 94.78], [9E9, 9E9, 9E9, 9E9, 9E9, 9E9]];
	VAR jointtarget CDP_3648 := [[-11.72, 36.33, 5.02, 0, 48.65, 96.92], [9E9, 9E9, 9E9, 9E9, 9E9, 9E9]];
	VAR jointtarget CDP_3649 := [[-11.78, 36.32, 5.03, 0, 48.65, 99.06], [9E9, 9E9, 9E9, 9E9, 9E9, 9E9]];
	VAR jointtarget CDP_3650 := [[-11.83, 36.31, 5.05, 0, 48.64, 101.2], [9E9, 9E9, 9E9, 9E9, 9E9, 9E9]];
	VAR jointtarget CDP_3651 := [[-11.89, 36.29, 5.08, 0, 48.63, 103.34], [9E9, 9E9, 9E9, 9E9, 9E9, 9E9]];
	VAR jointtarget CDP_3652 := [[-11.94, 36.28, 5.1, 0, 48.62, 105.48], [9E9, 9E9, 9E9, 9E9, 9E9, 9E9]];
	VAR jointtarget CDP_3653 := [[-11.99, 36.26, 5.14, 0, 48.6, 107.63], [9E9, 9E9, 9E9, 9E9, 9E9, 9E9]];
	VAR jointtarget CDP_3654 := [[-12.04, 36.24, 5.17, 0, 48.59, 109.77], [9E9, 9E9, 9E9, 9E9, 9E9, 9E9]];
	VAR jointtarget CDP_3655 := [[-12.09, 36.22, 5.21, 0, 48.57, 111.91], [9E9, 9E9, 9E9, 9E9, 9E9, 9E9]];
	VAR jointtarget CDP_3656 := [[-12.15, 36.19, 5.25, 0, 48.56, 114.05], [9E9, 9E9, 9E9, 9E9, 9E9, 9E9]];
	VAR jointtarget CDP_3657 := [[-12.19, 36.17, 5.3, 0, 48.54, 116.2], [9E9, 9E9, 9E9, 9E9, 9E9, 9E9]];
	VAR jointtarget CDP_3658 := [[-12.24, 36.14, 5.35, 0, 48.52, 118.34], [9E9, 9E9, 9E9, 9E9, 9E9, 9E9]];
	VAR jointtarget CDP_3659 := [[-12.29, 36.11, 5.4, 0, 48.49, 120.49], [9E9, 9E9, 9E9, 9E9, 9E9, 9E9]];
	VAR jointtarget CDP_3660 := [[-12.32, 36.09, 5.43, 0, 48.48, 121.56], [9E9, 9E9, 9E9, 9E9, 9E9, 9E9]];
	VAR jointtarget CDP_3661 := [[-12.35, 36.07, 5.47, 0, 48.47, 121.53], [9E9, 9E9, 9E9, 9E9, 9E9, 9E9]];
	VAR jointtarget CDP_3662 := [[-12.38, 36.05, 5.5, 0, 48.45, 121.5], [9E9, 9E9, 9E9, 9E9, 9E9, 9E9]];
	VAR jointtarget CDP_3663 := [[-12.41, 36.03, 5.53, 0, 48.44, 121.47], [9E9, 9E9, 9E9, 9E9, 9E9, 9E9]];
	VAR jointtarget CDP_3664 := [[-12.43, 36.01, 5.56, 0, 48.43, 121.44], [9E9, 9E9, 9E9, 9E9, 9E9, 9E9]];
	VAR jointtarget CDP_3665 := [[-12.46, 35.99, 5.6, 0, 48.41, 121.41], [9E9, 9E9, 9E9, 9E9, 9E9, 9E9]];
	VAR jointtarget CDP_3666 := [[-12.49, 35.97, 5.63, 0, 48.4, 121.39], [9E9, 9E9, 9E9, 9E9, 9E9, 9E9]];
	VAR jointtarget CDP_3667 := [[-12.52, 35.95, 5.66, 0, 48.39, 121.36], [9E9, 9E9, 9E9, 9E9, 9E9, 9E9]];
	VAR jointtarget CDP_3668 := [[-12.55, 35.93, 5.69, 0, 48.37, 121.33], [9E9, 9E9, 9E9, 9E9, 9E9, 9E9]];
	VAR jointtarget CDP_3669 := [[-12.58, 35.92, 5.73, 0, 48.36, 121.3], [9E9, 9E9, 9E9, 9E9, 9E9, 9E9]];
	VAR jointtarget CDP_3670 := [[-12.61, 35.9, 5.76, 0, 48.34, 121.27], [9E9, 9E9, 9E9, 9E9, 9E9, 9E9]];
	VAR jointtarget CDP_3671 := [[-12.63, 35.88, 5.79, 0, 48.33, 121.24], [9E9, 9E9, 9E9, 9E9, 9E9, 9E9]];
	VAR jointtarget CDP_3672 := [[-12.66, 35.86, 5.82, 0, 48.32, 121.21], [9E9, 9E9, 9E9, 9E9, 9E9, 9E9]];
	VAR jointtarget CDP_3673 := [[-12.69, 35.84, 5.86, 0, 48.3, 121.18], [9E9, 9E9, 9E9, 9E9, 9E9, 9E9]];
	VAR jointtarget CDP_3674 := [[-12.72, 35.82, 5.89, 0, 48.29, 121.16], [9E9, 9E9, 9E9, 9E9, 9E9, 9E9]];
	VAR jointtarget CDP_3675 := [[-12.75, 35.8, 5.92, 0, 48.28, 121.13], [9E9, 9E9, 9E9, 9E9, 9E9, 9E9]];
	VAR jointtarget CDP_3676 := [[-12.78, 35.78, 5.95, 0, 48.26, 121.1], [9E9, 9E9, 9E9, 9E9, 9E9, 9E9]];
	VAR jointtarget CDP_3677 := [[-12.81, 35.76, 5.98, 0, 48.25, 121.07], [9E9, 9E9, 9E9, 9E9, 9E9, 9E9]];
	VAR jointtarget CDP_3678 := [[-12.84, 35.75, 6.02, 0, 48.24, 121.04], [9E9, 9E9, 9E9, 9E9, 9E9, 9E9]];
	VAR jointtarget CDP_3679 := [[-12.86, 35.73, 6.05, 0, 48.22, 121.01], [9E9, 9E9, 9E9, 9E9, 9E9, 9E9]];
	VAR jointtarget CDP_3680 := [[-13.02, 35.65, 6.17, 0, 48.17, 114.17], [9E9, 9E9, 9E9, 9E9, 9E9, 9E9]];
	VAR jointtarget CDP_3681 := [[-13.18, 35.62, 6.23, 0, 48.15, 100.62], [9E9, 9E9, 9E9, 9E9, 9E9, 9E9]];
	VAR jointtarget CDP_3682 := [[-13.34, 35.63, 6.22, 0, 48.16, 87.07], [9E9, 9E9, 9E9, 9E9, 9E9, 9E9]];
	VAR jointtarget CDP_3683 := [[-13.5, 35.68, 6.13, 0, 48.19, 73.52], [9E9, 9E9, 9E9, 9E9, 9E9, 9E9]];
	VAR jointtarget CDP_3684 := [[-13.64, 35.77, 5.98, 0, 48.25, 59.99], [9E9, 9E9, 9E9, 9E9, 9E9, 9E9]];
	VAR jointtarget CDP_3685 := [[-13.76, 35.89, 5.77, 0, 48.34, 46.48], [9E9, 9E9, 9E9, 9E9, 9E9, 9E9]];
	VAR jointtarget CDP_3686 := [[-13.85, 36.04, 5.51, 0, 48.45, 33.01], [9E9, 9E9, 9E9, 9E9, 9E9, 9E9]];
	VAR jointtarget CDP_3687 := [[-13.91, 36.21, 5.22, 0, 48.57, 19.56], [9E9, 9E9, 9E9, 9E9, 9E9, 9E9]];
	VAR jointtarget CDP_3688 := [[-13.92, 36.39, 4.92, 0, 48.7, 6.16], [9E9, 9E9, 9E9, 9E9, 9E9, 9E9]];
	VAR jointtarget CDP_3689 := [[-13.9, 36.57, 4.61, 0, 48.82, -7.21], [9E9, 9E9, 9E9, 9E9, 9E9, 9E9]];
	VAR jointtarget CDP_3690 := [[-13.85, 36.73, 4.32, 0, 48.94, -20.54], [9E9, 9E9, 9E9, 9E9, 9E9, 9E9]];
	VAR jointtarget CDP_3691 := [[-13.76, 36.88, 4.07, 0, 49.05, -33.84], [9E9, 9E9, 9E9, 9E9, 9E9, 9E9]];
	VAR jointtarget CDP_3692 := [[-13.64, 37.01, 3.85, 0, 49.14, -47.11], [9E9, 9E9, 9E9, 9E9, 9E9, 9E9]];
	VAR jointtarget CDP_3693 := [[-13.5, 37.09, 3.7, 0, 49.2, -60.35], [9E9, 9E9, 9E9, 9E9, 9E9, 9E9]];
	VAR jointtarget CDP_3694 := [[-13.34, 37.15, 3.61, 0, 49.24, -73.59], [9E9, 9E9, 9E9, 9E9, 9E9, 9E9]];
	VAR jointtarget CDP_3695 := [[-13.18, 37.16, 3.6, 0, 49.25, -86.81], [9E9, 9E9, 9E9, 9E9, 9E9, 9E9]];
	VAR jointtarget CDP_3696 := [[-13.02, 37.12, 3.65, 0, 49.22, -100.04], [9E9, 9E9, 9E9, 9E9, 9E9, 9E9]];
	VAR jointtarget CDP_3697 := [[-12.88, 37.05, 3.77, 0, 49.17, -113.28], [9E9, 9E9, 9E9, 9E9, 9E9, 9E9]];
	VAR jointtarget CDP_3698 := [[-12.75, 36.94, 3.96, 0, 49.1, -126.54], [9E9, 9E9, 9E9, 9E9, 9E9, 9E9]];
	VAR jointtarget CDP_3699 := [[-12.64, 36.81, 4.2, 0, 49, -139.82], [9E9, 9E9, 9E9, 9E9, 9E9, 9E9]];
	VAR jointtarget CDP_3700 := [[-12.62, 36.77, 4.27, 0, 48.97, -146.49], [9E9, 9E9, 9E9, 9E9, 9E9, 9E9]];
	VAR jointtarget CDP_3701 := [[-12.59, 36.72, 4.34, 0, 48.94, -146.47], [9E9, 9E9, 9E9, 9E9, 9E9, 9E9]];
	VAR jointtarget CDP_3702 := [[-12.57, 36.68, 4.41, 0, 48.91, -146.44], [9E9, 9E9, 9E9, 9E9, 9E9, 9E9]];
	VAR jointtarget CDP_3703 := [[-12.54, 36.64, 4.48, 0, 48.88, -146.42], [9E9, 9E9, 9E9, 9E9, 9E9, 9E9]];
	VAR jointtarget CDP_3704 := [[-12.52, 36.6, 4.55, 0, 48.85, -146.4], [9E9, 9E9, 9E9, 9E9, 9E9, 9E9]];
	VAR jointtarget CDP_3705 := [[-12.49, 36.56, 4.62, 0, 48.82, -146.37], [9E9, 9E9, 9E9, 9E9, 9E9, 9E9]];
	VAR jointtarget CDP_3706 := [[-12.47, 36.52, 4.69, 0, 48.79, -146.35], [9E9, 9E9, 9E9, 9E9, 9E9, 9E9]];
	VAR jointtarget CDP_3707 := [[-12.44, 36.48, 4.76, 0, 48.76, -146.32], [9E9, 9E9, 9E9, 9E9, 9E9, 9E9]];
	VAR jointtarget CDP_3708 := [[-12.42, 36.44, 4.83, 0, 48.73, -146.3], [9E9, 9E9, 9E9, 9E9, 9E9, 9E9]];
	VAR jointtarget CDP_3709 := [[-12.39, 36.39, 4.9, 0, 48.7, -146.27], [9E9, 9E9, 9E9, 9E9, 9E9, 9E9]];
	VAR jointtarget CDP_3710 := [[-12.37, 36.35, 4.97, 0, 48.67, -146.25], [9E9, 9E9, 9E9, 9E9, 9E9, 9E9]];
	VAR jointtarget CDP_3711 := [[-12.34, 36.31, 5.05, 0, 48.64, -146.22], [9E9, 9E9, 9E9, 9E9, 9E9, 9E9]];
	VAR jointtarget CDP_3712 := [[-12.32, 36.27, 5.12, 0, 48.61, -146.2], [9E9, 9E9, 9E9, 9E9, 9E9, 9E9]];
	VAR jointtarget CDP_3713 := [[-12.29, 36.23, 5.19, 0, 48.58, -146.17], [9E9, 9E9, 9E9, 9E9, 9E9, 9E9]];
	VAR jointtarget CDP_3714 := [[-12.27, 36.19, 5.26, 0, 48.55, -146.15], [9E9, 9E9, 9E9, 9E9, 9E9, 9E9]];
	VAR jointtarget CDP_3715 := [[-12.24, 36.15, 5.33, 0, 48.52, -146.12], [9E9, 9E9, 9E9, 9E9, 9E9, 9E9]];
	VAR jointtarget CDP_3716 := [[-12.22, 36.11, 5.4, 0, 48.5, -146.1], [9E9, 9E9, 9E9, 9E9, 9E9, 9E9]];
	VAR jointtarget CDP_3717 := [[-12.19, 36.07, 5.47, 0, 48.47, -146.07], [9E9, 9E9, 9E9, 9E9, 9E9, 9E9]];
	VAR jointtarget CDP_3718 := [[-12.17, 36.03, 5.54, 0, 48.44, -146.05], [9E9, 9E9, 9E9, 9E9, 9E9, 9E9]];
	VAR jointtarget CDP_3719 := [[-12.14, 35.99, 5.61, 0, 48.41, -146.02], [9E9, 9E9, 9E9, 9E9, 9E9, 9E9]];
	VAR jointtarget CDP_3720 := [[-12.14, 35.97, 5.63, 0, 48.4, -145.46], [9E9, 9E9, 9E9, 9E9, 9E9, 9E9]];
	VAR jointtarget CDP_3721 := [[-12.13, 35.96, 5.65, 0, 48.39, -144.35], [9E9, 9E9, 9E9, 9E9, 9E9, 9E9]];
	VAR jointtarget CDP_3722 := [[-12.12, 35.95, 5.67, 0, 48.38, -143.24], [9E9, 9E9, 9E9, 9E9, 9E9, 9E9]];
	VAR jointtarget CDP_3723 := [[-12.11, 35.94, 5.69, 0, 48.37, -142.13], [9E9, 9E9, 9E9, 9E9, 9E9, 9E9]];
	VAR jointtarget CDP_3724 := [[-12.1, 35.92, 5.71, 0, 48.37, -141.01], [9E9, 9E9, 9E9, 9E9, 9E9, 9E9]];
	VAR jointtarget CDP_3725 := [[-12.09, 35.91, 5.73, 0, 48.36, -139.9], [9E9, 9E9, 9E9, 9E9, 9E9, 9E9]];
	VAR jointtarget CDP_3726 := [[-12.08, 35.9, 5.75, 0, 48.35, -138.79], [9E9, 9E9, 9E9, 9E9, 9E9, 9E9]];
	VAR jointtarget CDP_3727 := [[-12.07, 35.89, 5.77, 0, 48.34, -137.68], [9E9, 9E9, 9E9, 9E9, 9E9, 9E9]];
	VAR jointtarget CDP_3728 := [[-12.06, 35.88, 5.79, 0, 48.33, -136.56], [9E9, 9E9, 9E9, 9E9, 9E9, 9E9]];
	VAR jointtarget CDP_3729 := [[-12.05, 35.87, 5.81, 0, 48.33, -135.45], [9E9, 9E9, 9E9, 9E9, 9E9, 9E9]];
	VAR jointtarget CDP_3730 := [[-12.04, 35.86, 5.83, 0, 48.32, -134.34], [9E9, 9E9, 9E9, 9E9, 9E9, 9E9]];
	VAR jointtarget CDP_3731 := [[-12.03, 35.85, 5.84, 0, 48.31, -133.22], [9E9, 9E9, 9E9, 9E9, 9E9, 9E9]];
	VAR jointtarget CDP_3732 := [[-12.02, 35.83, 5.86, 0, 48.3, -132.11], [9E9, 9E9, 9E9, 9E9, 9E9, 9E9]];
	VAR jointtarget CDP_3733 := [[-12.01, 35.82, 5.88, 0, 48.3, -130.99], [9E9, 9E9, 9E9, 9E9, 9E9, 9E9]];
	VAR jointtarget CDP_3734 := [[-12, 35.81, 5.89, 0, 48.29, -129.88], [9E9, 9E9, 9E9, 9E9, 9E9, 9E9]];
	VAR jointtarget CDP_3735 := [[-11.99, 35.8, 5.91, 0, 48.29, -128.76], [9E9, 9E9, 9E9, 9E9, 9E9, 9E9]];
	VAR jointtarget CDP_3736 := [[-11.98, 35.79, 5.93, 0, 48.28, -127.65], [9E9, 9E9, 9E9, 9E9, 9E9, 9E9]];
	VAR jointtarget CDP_3737 := [[-11.97, 35.79, 5.94, 0, 48.27, -126.53], [9E9, 9E9, 9E9, 9E9, 9E9, 9E9]];
	VAR jointtarget CDP_3738 := [[-11.96, 35.78, 5.96, 0, 48.27, -125.42], [9E9, 9E9, 9E9, 9E9, 9E9, 9E9]];
	VAR jointtarget CDP_3739 := [[-11.95, 35.77, 5.97, 0, 48.26, -124.3], [9E9, 9E9, 9E9, 9E9, 9E9, 9E9]];
	VAR jointtarget CDP_3740 := [[-11.94, 35.76, 5.98, 0, 48.26, -123.74], [9E9, 9E9, 9E9, 9E9, 9E9, 9E9]];
	VAR jointtarget CDP_3741 := [[-11.93, 35.75, 6, 0, 48.25, -123.73], [9E9, 9E9, 9E9, 9E9, 9E9, 9E9]];
	VAR jointtarget CDP_3742 := [[-11.92, 35.74, 6.01, 0, 48.25, -123.72], [9E9, 9E9, 9E9, 9E9, 9E9, 9E9]];
	VAR jointtarget CDP_3743 := [[-11.9, 35.74, 6.02, 0, 48.24, -123.71], [9E9, 9E9, 9E9, 9E9, 9E9, 9E9]];
	VAR jointtarget CDP_3744 := [[-11.89, 35.73, 6.03, 0, 48.24, -123.7], [9E9, 9E9, 9E9, 9E9, 9E9, 9E9]];
	VAR jointtarget CDP_3745 := [[-11.88, 35.72, 6.05, 0, 48.23, -123.69], [9E9, 9E9, 9E9, 9E9, 9E9, 9E9]];
	VAR jointtarget CDP_3746 := [[-11.87, 35.71, 6.06, 0, 48.23, -123.68], [9E9, 9E9, 9E9, 9E9, 9E9, 9E9]];
	VAR jointtarget CDP_3747 := [[-11.86, 35.7, 6.07, 0, 48.22, -123.66], [9E9, 9E9, 9E9, 9E9, 9E9, 9E9]];
	VAR jointtarget CDP_3748 := [[-11.85, 35.7, 6.09, 0, 48.22, -123.65], [9E9, 9E9, 9E9, 9E9, 9E9, 9E9]];
	VAR jointtarget CDP_3749 := [[-11.84, 35.69, 6.1, 0, 48.21, -123.64], [9E9, 9E9, 9E9, 9E9, 9E9, 9E9]];
	VAR jointtarget CDP_3750 := [[-11.83, 35.68, 6.11, 0, 48.21, -123.63], [9E9, 9E9, 9E9, 9E9, 9E9, 9E9]];
	VAR jointtarget CDP_3751 := [[-11.82, 35.67, 6.12, 0, 48.2, -123.62], [9E9, 9E9, 9E9, 9E9, 9E9, 9E9]];
	VAR jointtarget CDP_3752 := [[-11.81, 35.66, 6.14, 0, 48.2, -123.61], [9E9, 9E9, 9E9, 9E9, 9E9, 9E9]];
	VAR jointtarget CDP_3753 := [[-11.8, 35.66, 6.15, 0, 48.19, -123.6], [9E9, 9E9, 9E9, 9E9, 9E9, 9E9]];
	VAR jointtarget CDP_3754 := [[-11.79, 35.65, 6.16, 0, 48.19, -123.59], [9E9, 9E9, 9E9, 9E9, 9E9, 9E9]];
	VAR jointtarget CDP_3755 := [[-11.78, 35.64, 6.17, 0, 48.18, -123.58], [9E9, 9E9, 9E9, 9E9, 9E9, 9E9]];
	VAR jointtarget CDP_3756 := [[-11.77, 35.63, 6.19, 0, 48.18, -123.57], [9E9, 9E9, 9E9, 9E9, 9E9, 9E9]];
	VAR jointtarget CDP_3757 := [[-11.76, 35.62, 6.2, 0, 48.18, -123.56], [9E9, 9E9, 9E9, 9E9, 9E9, 9E9]];
	VAR jointtarget CDP_3758 := [[-11.75, 35.62, 6.21, 0, 48.17, -123.55], [9E9, 9E9, 9E9, 9E9, 9E9, 9E9]];
	VAR jointtarget CDP_3759 := [[-11.74, 35.61, 6.23, 0, 48.17, -123.54], [9E9, 9E9, 9E9, 9E9, 9E9, 9E9]];
	VAR jointtarget CDP_3760 := [[-10.65, 35.38, 6.62, 0, 48, -100.65], [9E9, 9E9, 9E9, 9E9, 9E9, 9E9]];
	VAR jointtarget CDP_3761 := [[-9.55, 35.17, 6.98, 0, 47.85, -99.55], [9E9, 9E9, 9E9, 9E9, 9E9, 9E9]];
	VAR jointtarget CDP_3762 := [[-8.44, 34.98, 7.3, 0, 47.72, -98.44], [9E9, 9E9, 9E9, 9E9, 9E9, 9E9]];
	VAR jointtarget CDP_3763 := [[-7.33, 34.82, 7.58, 0, 47.61, -97.33], [9E9, 9E9, 9E9, 9E9, 9E9, 9E9]];
	VAR jointtarget CDP_3764 := [[-6.21, 34.68, 7.81, 0, 47.51, -96.21], [9E9, 9E9, 9E9, 9E9, 9E9, 9E9]];
	VAR jointtarget CDP_3765 := [[-5.09, 34.56, 8.01, 0, 47.43, -95.09], [9E9, 9E9, 9E9, 9E9, 9E9, 9E9]];
	VAR jointtarget CDP_3766 := [[-3.96, 34.46, 8.17, 0, 47.36, -93.96], [9E9, 9E9, 9E9, 9E9, 9E9, 9E9]];
	VAR jointtarget CDP_3767 := [[-2.83, 34.39, 8.29, 0, 47.31, -92.83], [9E9, 9E9, 9E9, 9E9, 9E9, 9E9]];
	VAR jointtarget CDP_3768 := [[-1.7, 34.35, 8.37, 0, 47.28, -91.7], [9E9, 9E9, 9E9, 9E9, 9E9, 9E9]];
	VAR jointtarget CDP_3769 := [[-0.56, 34.32, 8.41, 0, 47.26, -90.56], [9E9, 9E9, 9E9, 9E9, 9E9, 9E9]];
	VAR jointtarget CDP_3770 := [[0.57, 34.32, 8.41, 0, 47.26, -89.43], [9E9, 9E9, 9E9, 9E9, 9E9, 9E9]];
	VAR jointtarget CDP_3771 := [[1.7, 34.35, 8.37, 0, 47.28, -88.3], [9E9, 9E9, 9E9, 9E9, 9E9, 9E9]];
	VAR jointtarget CDP_3772 := [[2.84, 34.4, 8.29, 0, 47.31, -87.16], [9E9, 9E9, 9E9, 9E9, 9E9, 9E9]];
	VAR jointtarget CDP_3773 := [[3.97, 34.47, 8.17, 0, 47.36, -86.03], [9E9, 9E9, 9E9, 9E9, 9E9, 9E9]];
	VAR jointtarget CDP_3774 := [[5.09, 34.56, 8.01, 0, 47.43, -84.91], [9E9, 9E9, 9E9, 9E9, 9E9, 9E9]];
	VAR jointtarget CDP_3775 := [[6.22, 34.68, 7.81, 0, 47.51, -83.78], [9E9, 9E9, 9E9, 9E9, 9E9, 9E9]];
	VAR jointtarget CDP_3776 := [[7.34, 34.82, 7.57, 0, 47.61, -82.66], [9E9, 9E9, 9E9, 9E9, 9E9, 9E9]];
	VAR jointtarget CDP_3777 := [[8.45, 34.98, 7.3, 0, 47.72, -81.55], [9E9, 9E9, 9E9, 9E9, 9E9, 9E9]];
	VAR jointtarget CDP_3778 := [[9.56, 35.17, 6.98, 0, 47.85, -80.44], [9E9, 9E9, 9E9, 9E9, 9E9, 9E9]];
	VAR jointtarget CDP_3779 := [[10.65, 35.38, 6.62, 0, 48, -79.35], [9E9, 9E9, 9E9, 9E9, 9E9, 9E9]];
	VAR jointtarget CDP_3780 := [[10.71, 35.39, 6.6, 0, 48.01, -78.19], [9E9, 9E9, 9E9, 9E9, 9E9, 9E9]];
	VAR jointtarget CDP_3781 := [[10.76, 35.4, 6.57, 0, 48.02, -75.95], [9E9, 9E9, 9E9, 9E9, 9E9, 9E9]];
	VAR jointtarget CDP_3782 := [[10.82, 35.42, 6.54, 0, 48.03, -73.7], [9E9, 9E9, 9E9, 9E9, 9E9, 9E9]];
	VAR jointtarget CDP_3783 := [[10.87, 35.44, 6.51, 0, 48.05, -71.45], [9E9, 9E9, 9E9, 9E9, 9E9, 9E9]];
	VAR jointtarget CDP_3784 := [[10.92, 35.46, 6.48, 0, 48.06, -69.2], [9E9, 9E9, 9E9, 9E9, 9E9, 9E9]];
	VAR jointtarget CDP_3785 := [[10.97, 35.49, 6.44, 0, 48.08, -66.96], [9E9, 9E9, 9E9, 9E9, 9E9, 9E9]];
	VAR jointtarget CDP_3786 := [[11.03, 35.51, 6.39, 0, 48.1, -64.72], [9E9, 9E9, 9E9, 9E9, 9E9, 9E9]];
	VAR jointtarget CDP_3787 := [[11.07, 35.54, 6.34, 0, 48.12, -62.47], [9E9, 9E9, 9E9, 9E9, 9E9, 9E9]];
	VAR jointtarget CDP_3788 := [[11.12, 35.57, 6.29, 0, 48.14, -60.23], [9E9, 9E9, 9E9, 9E9, 9E9, 9E9]];
	VAR jointtarget CDP_3789 := [[11.17, 35.6, 6.24, 0, 48.16, -57.99], [9E9, 9E9, 9E9, 9E9, 9E9, 9E9]];
	VAR jointtarget CDP_3790 := [[11.22, 35.63, 6.18, 0, 48.18, -55.75], [9E9, 9E9, 9E9, 9E9, 9E9, 9E9]];
	VAR jointtarget CDP_3791 := [[11.26, 35.67, 6.12, 0, 48.21, -53.51], [9E9, 9E9, 9E9, 9E9, 9E9, 9E9]];
	VAR jointtarget CDP_3792 := [[11.3, 35.71, 6.06, 0, 48.24, -51.27], [9E9, 9E9, 9E9, 9E9, 9E9, 9E9]];
	VAR jointtarget CDP_3793 := [[11.35, 35.75, 5.99, 0, 48.26, -49.04], [9E9, 9E9, 9E9, 9E9, 9E9, 9E9]];
	VAR jointtarget CDP_3794 := [[11.39, 35.79, 5.92, 0, 48.29, -46.8], [9E9, 9E9, 9E9, 9E9, 9E9, 9E9]];
	VAR jointtarget CDP_3795 := [[11.43, 35.83, 5.84, 0, 48.32, -44.57], [9E9, 9E9, 9E9, 9E9, 9E9, 9E9]];
	VAR jointtarget CDP_3796 := [[11.46, 35.88, 5.77, 0, 48.36, -42.34], [9E9, 9E9, 9E9, 9E9, 9E9, 9E9]];
	VAR jointtarget CDP_3797 := [[11.5, 35.92, 5.69, 0, 48.39, -40.11], [9E9, 9E9, 9E9, 9E9, 9E9, 9E9]];
	VAR jointtarget CDP_3798 := [[11.53, 35.97, 5.61, 0, 48.42, -37.88], [9E9, 9E9, 9E9, 9E9, 9E9, 9E9]];
	VAR jointtarget CDP_3799 := [[11.57, 36.02, 5.52, 0, 48.46, -35.65], [9E9, 9E9, 9E9, 9E9, 9E9, 9E9]];
	VAR jointtarget CDP_3800 := [[11.59, 36.05, 5.47, 0, 48.48, -34.54], [9E9, 9E9, 9E9, 9E9, 9E9, 9E9]];
	VAR jointtarget CDP_3801 := [[11.6, 36.08, 5.42, 0, 48.5, -34.52], [9E9, 9E9, 9E9, 9E9, 9E9, 9E9]];
	VAR jointtarget CDP_3802 := [[11.62, 36.11, 5.37, 0, 48.52, -34.5], [9E9, 9E9, 9E9, 9E9, 9E9, 9E9]];
	VAR jointtarget CDP_3803 := [[11.64, 36.14, 5.32, 0, 48.54, -34.48], [9E9, 9E9, 9E9, 9E9, 9E9, 9E9]];
	VAR jointtarget CDP_3804 := [[11.66, 36.17, 5.26, 0, 48.56, -34.46], [9E9, 9E9, 9E9, 9E9, 9E9, 9E9]];
	VAR jointtarget CDP_3805 := [[11.68, 36.2, 5.21, 0, 48.59, -34.44], [9E9, 9E9, 9E9, 9E9, 9E9, 9E9]];
	VAR jointtarget CDP_3806 := [[11.7, 36.23, 5.16, 0, 48.61, -34.42], [9E9, 9E9, 9E9, 9E9, 9E9, 9E9]];
	VAR jointtarget CDP_3807 := [[11.72, 36.26, 5.11, 0, 48.63, -34.41], [9E9, 9E9, 9E9, 9E9, 9E9, 9E9]];
	VAR jointtarget CDP_3808 := [[11.74, 36.29, 5.06, 0, 48.65, -34.39], [9E9, 9E9, 9E9, 9E9, 9E9, 9E9]];
	VAR jointtarget CDP_3809 := [[11.76, 36.32, 5.01, 0, 48.67, -34.37], [9E9, 9E9, 9E9, 9E9, 9E9, 9E9]];
	VAR jointtarget CDP_3810 := [[11.77, 36.35, 4.95, 0, 48.69, -34.35], [9E9, 9E9, 9E9, 9E9, 9E9, 9E9]];
	VAR jointtarget CDP_3811 := [[11.79, 36.38, 4.9, 0, 48.72, -34.33], [9E9, 9E9, 9E9, 9E9, 9E9, 9E9]];
	VAR jointtarget CDP_3812 := [[11.81, 36.41, 4.85, 0, 48.74, -34.31], [9E9, 9E9, 9E9, 9E9, 9E9, 9E9]];
	VAR jointtarget CDP_3813 := [[11.83, 36.44, 4.8, 0, 48.76, -34.29], [9E9, 9E9, 9E9, 9E9, 9E9, 9E9]];
	VAR jointtarget CDP_3814 := [[11.85, 36.47, 4.75, 0, 48.78, -34.27], [9E9, 9E9, 9E9, 9E9, 9E9, 9E9]];
	VAR jointtarget CDP_3815 := [[11.87, 36.5, 4.69, 0, 48.8, -34.26], [9E9, 9E9, 9E9, 9E9, 9E9, 9E9]];
	VAR jointtarget CDP_3816 := [[11.89, 36.53, 4.64, 0, 48.82, -34.24], [9E9, 9E9, 9E9, 9E9, 9E9, 9E9]];
	VAR jointtarget CDP_3817 := [[11.91, 36.56, 4.59, 0, 48.85, -34.22], [9E9, 9E9, 9E9, 9E9, 9E9, 9E9]];
	VAR jointtarget CDP_3818 := [[11.92, 36.59, 4.54, 0, 48.87, -34.2], [9E9, 9E9, 9E9, 9E9, 9E9, 9E9]];
	VAR jointtarget CDP_3819 := [[11.94, 36.62, 4.49, 0, 48.89, -34.18], [9E9, 9E9, 9E9, 9E9, 9E9, 9E9]];
	VAR jointtarget CDP_3820 := [[12.05, 36.76, 4.25, 0, 48.99, -40.77], [9E9, 9E9, 9E9, 9E9, 9E9, 9E9]];
	VAR jointtarget CDP_3821 := [[12.18, 36.87, 4.07, 0, 49.06, -54.03], [9E9, 9E9, 9E9, 9E9, 9E9, 9E9]];
	VAR jointtarget CDP_3822 := [[12.33, 36.94, 3.95, 0, 49.11, -67.26], [9E9, 9E9, 9E9, 9E9, 9E9, 9E9]];
	VAR jointtarget CDP_3823 := [[12.49, 36.97, 3.9, 0, 49.14, -80.49], [9E9, 9E9, 9E9, 9E9, 9E9, 9E9]];
	VAR jointtarget CDP_3824 := [[12.65, 36.95, 3.92, 0, 49.13, -93.72], [9E9, 9E9, 9E9, 9E9, 9E9, 9E9]];
	VAR jointtarget CDP_3825 := [[12.8, 36.9, 4.01, 0, 49.09, -106.95], [9E9, 9E9, 9E9, 9E9, 9E9, 9E9]];
	VAR jointtarget CDP_3826 := [[12.94, 36.81, 4.17, 0, 49.02, -120.2], [9E9, 9E9, 9E9, 9E9, 9E9, 9E9]];
	VAR jointtarget CDP_3827 := [[13.06, 36.69, 4.38, 0, 48.93, -133.47], [9E9, 9E9, 9E9, 9E9, 9E9, 9E9]];
	VAR jointtarget CDP_3828 := [[13.15, 36.54, 4.64, 0, 48.83, -146.77], [9E9, 9E9, 9E9, 9E9, 9E9, 9E9]];
	VAR jointtarget CDP_3829 := [[13.2, 36.37, 4.93, 0, 48.71, -160.1], [9E9, 9E9, 9E9, 9E9, 9E9, 9E9]];
	VAR jointtarget CDP_3830 := [[13.22, 36.19, 5.23, 0, 48.58, -173.47], [9E9, 9E9, 9E9, 9E9, 9E9, 9E9]];
	VAR jointtarget CDP_3831 := [[13.2, 36.01, 5.54, 0, 48.45, -186.88], [9E9, 9E9, 9E9, 9E9, 9E9, 9E9]];
	VAR jointtarget CDP_3832 := [[13.15, 35.84, 5.82, 0, 48.33, -200.32], [9E9, 9E9, 9E9, 9E9, 9E9, 9E9]];
	VAR jointtarget CDP_3833 := [[13.06, 35.7, 6.08, 0, 48.23, -213.8], [9E9, 9E9, 9E9, 9E9, 9E9, 9E9]];
	VAR jointtarget CDP_3834 := [[12.93, 35.57, 6.28, 0, 48.14, -227.31], [9E9, 9E9, 9E9, 9E9, 9E9, 9E9]];
	VAR jointtarget CDP_3835 := [[12.79, 35.49, 6.43, 0, 48.08, -240.84], [9E9, 9E9, 9E9, 9E9, 9E9, 9E9]];
	VAR jointtarget CDP_3836 := [[12.63, 35.44, 6.51, 0, 48.05, -254.39], [9E9, 9E9, 9E9, 9E9, 9E9, 9E9]];
	VAR jointtarget CDP_3837 := [[12.47, 35.43, 6.53, 0, 48.04, -267.94], [9E9, 9E9, 9E9, 9E9, 9E9, 9E9]];
	VAR jointtarget CDP_3838 := [[12.3, 35.47, 6.47, 0, 48.07, -281.49], [9E9, 9E9, 9E9, 9E9, 9E9, 9E9]];
	VAR jointtarget CDP_3839 := [[12.15, 35.54, 6.34, 0, 48.12, -295.03], [9E9, 9E9, 9E9, 9E9, 9E9, 9E9]];
	VAR jointtarget CDP_3840 := [[12.13, 35.56, 6.31, 0, 48.13, -301.75], [9E9, 9E9, 9E9, 9E9, 9E9, 9E9]];
	VAR jointtarget CDP_3841 := [[12.1, 35.58, 6.27, 0, 48.15, -301.78], [9E9, 9E9, 9E9, 9E9, 9E9, 9E9]];
	VAR jointtarget CDP_3842 := [[12.07, 35.6, 6.24, 0, 48.16, -301.81], [9E9, 9E9, 9E9, 9E9, 9E9, 9E9]];
	VAR jointtarget CDP_3843 := [[12.04, 35.62, 6.21, 0, 48.17, -301.84], [9E9, 9E9, 9E9, 9E9, 9E9, 9E9]];
	VAR jointtarget CDP_3844 := [[12.01, 35.64, 6.17, 0, 48.19, -301.87], [9E9, 9E9, 9E9, 9E9, 9E9, 9E9]];
	VAR jointtarget CDP_3845 := [[11.98, 35.66, 6.14, 0, 48.2, -301.89], [9E9, 9E9, 9E9, 9E9, 9E9, 9E9]];
	VAR jointtarget CDP_3846 := [[11.95, 35.68, 6.11, 0, 48.21, -301.92], [9E9, 9E9, 9E9, 9E9, 9E9, 9E9]];
	VAR jointtarget CDP_3847 := [[11.92, 35.7, 6.08, 0, 48.23, -301.95], [9E9, 9E9, 9E9, 9E9, 9E9, 9E9]];
	VAR jointtarget CDP_3848 := [[11.9, 35.72, 6.04, 0, 48.24, -301.98], [9E9, 9E9, 9E9, 9E9, 9E9, 9E9]];
	VAR jointtarget CDP_3849 := [[11.87, 35.74, 6.01, 0, 48.26, -302.01], [9E9, 9E9, 9E9, 9E9, 9E9, 9E9]];
	VAR jointtarget CDP_3850 := [[11.84, 35.75, 5.98, 0, 48.27, -302.04], [9E9, 9E9, 9E9, 9E9, 9E9, 9E9]];
	VAR jointtarget CDP_3851 := [[11.81, 35.77, 5.94, 0, 48.28, -302.07], [9E9, 9E9, 9E9, 9E9, 9E9, 9E9]];
	VAR jointtarget CDP_3852 := [[11.78, 35.79, 5.91, 0, 48.3, -302.09], [9E9, 9E9, 9E9, 9E9, 9E9, 9E9]];
	VAR jointtarget CDP_3853 := [[11.75, 35.81, 5.88, 0, 48.31, -302.12], [9E9, 9E9, 9E9, 9E9, 9E9, 9E9]];
	VAR jointtarget CDP_3854 := [[11.73, 35.83, 5.84, 0, 48.32, -302.15], [9E9, 9E9, 9E9, 9E9, 9E9, 9E9]];
	VAR jointtarget CDP_3855 := [[11.7, 35.85, 5.81, 0, 48.34, -302.18], [9E9, 9E9, 9E9, 9E9, 9E9, 9E9]];
	VAR jointtarget CDP_3856 := [[11.67, 35.87, 5.78, 0, 48.35, -302.21], [9E9, 9E9, 9E9, 9E9, 9E9, 9E9]];
	VAR jointtarget CDP_3857 := [[11.64, 35.89, 5.74, 0, 48.37, -302.24], [9E9, 9E9, 9E9, 9E9, 9E9, 9E9]];
	VAR jointtarget CDP_3858 := [[11.61, 35.91, 5.71, 0, 48.38, -302.27], [9E9, 9E9, 9E9, 9E9, 9E9, 9E9]];
	VAR jointtarget CDP_3859 := [[11.58, 35.93, 5.68, 0, 48.39, -302.29], [9E9, 9E9, 9E9, 9E9, 9E9, 9E9]];
	VAR jointtarget CDP_3860 := [[11.54, 35.96, 5.62, 0, 48.42, -301.24], [9E9, 9E9, 9E9, 9E9, 9E9, 9E9]];
	VAR jointtarget CDP_3861 := [[11.49, 35.99, 5.57, 0, 48.44, -299.1], [9E9, 9E9, 9E9, 9E9, 9E9, 9E9]];
	VAR jointtarget CDP_3862 := [[11.44, 36.02, 5.53, 0, 48.46, -296.95], [9E9, 9E9, 9E9, 9E9, 9E9, 9E9]];
	VAR jointtarget CDP_3863 := [[11.39, 36.04, 5.48, 0, 48.47, -294.81], [9E9, 9E9, 9E9, 9E9, 9E9, 9E9]];
	VAR jointtarget CDP_3864 := [[11.34, 36.07, 5.44, 0, 48.49, -292.67], [9E9, 9E9, 9E9, 9E9, 9E9, 9E9]];
	VAR jointtarget CDP_3865 := [[11.28, 36.09, 5.41, 0, 48.51, -290.53], [9E9, 9E9, 9E9, 9E9, 9E9, 9E9]];
	VAR jointtarget CDP_3866 := [[11.23, 36.11, 5.37, 0, 48.52, -288.38], [9E9, 9E9, 9E9, 9E9, 9E9, 9E9]];
	VAR jointtarget CDP_3867 := [[11.18, 36.12, 5.35, 0, 48.53, -286.24], [9E9, 9E9, 9E9, 9E9, 9E9, 9E9]];
	VAR jointtarget CDP_3868 := [[11.13, 36.14, 5.32, 0, 48.54, -284.1], [9E9, 9E9, 9E9, 9E9, 9E9, 9E9]];
	VAR jointtarget CDP_3869 := [[11.07, 36.15, 5.3, 0, 48.55, -281.96], [9E9, 9E9, 9E9, 9E9, 9E9, 9E9]];
	VAR jointtarget CDP_3870 := [[11.02, 36.16, 5.28, 0, 48.56, -279.82], [9E9, 9E9, 9E9, 9E9, 9E9, 9E9]];
	VAR jointtarget CDP_3871 := [[10.96, 36.17, 5.27, 0, 48.56, -277.69], [9E9, 9E9, 9E9, 9E9, 9E9, 9E9]];
	VAR jointtarget CDP_3872 := [[10.91, 36.17, 5.26, 0, 48.57, -275.55], [9E9, 9E9, 9E9, 9E9, 9E9, 9E9]];
	VAR jointtarget CDP_3873 := [[10.85, 36.18, 5.25, 0, 48.57, -273.41], [9E9, 9E9, 9E9, 9E9, 9E9, 9E9]];
	VAR jointtarget CDP_3874 := [[10.8, 36.18, 5.25, 0, 48.57, -271.27], [9E9, 9E9, 9E9, 9E9, 9E9, 9E9]];
	VAR jointtarget CDP_3875 := [[10.74, 36.18, 5.25, 0, 48.57, -269.13], [9E9, 9E9, 9E9, 9E9, 9E9, 9E9]];
	VAR jointtarget CDP_3876 := [[10.69, 36.18, 5.26, 0, 48.57, -266.99], [9E9, 9E9, 9E9, 9E9, 9E9, 9E9]];
	VAR jointtarget CDP_3877 := [[10.63, 36.17, 5.27, 0, 48.56, -264.85], [9E9, 9E9, 9E9, 9E9, 9E9, 9E9]];
	VAR jointtarget CDP_3878 := [[10.58, 36.16, 5.28, 0, 48.56, -262.71], [9E9, 9E9, 9E9, 9E9, 9E9, 9E9]];
	VAR jointtarget CDP_3879 := [[10.52, 36.15, 5.3, 0, 48.55, -260.58], [9E9, 9E9, 9E9, 9E9, 9E9, 9E9]];
	VAR jointtarget CDP_3880 := [[9.44, 35.95, 5.65, 0, 48.4, -260.56], [9E9, 9E9, 9E9, 9E9, 9E9, 9E9]];
	VAR jointtarget CDP_3881 := [[8.36, 35.76, 5.97, 0, 48.27, -261.64], [9E9, 9E9, 9E9, 9E9, 9E9, 9E9]];
	VAR jointtarget CDP_3882 := [[7.27, 35.6, 6.24, 0, 48.16, -262.73], [9E9, 9E9, 9E9, 9E9, 9E9, 9E9]];
	VAR jointtarget CDP_3883 := [[6.17, 35.46, 6.48, 0, 48.06, -263.83], [9E9, 9E9, 9E9, 9E9, 9E9, 9E9]];
	VAR jointtarget CDP_3884 := [[5.07, 35.34, 6.68, 0, 47.98, -264.93], [9E9, 9E9, 9E9, 9E9, 9E9, 9E9]];
	VAR jointtarget CDP_3885 := [[3.97, 35.25, 6.84, 0, 47.91, -266.03], [9E9, 9E9, 9E9, 9E9, 9E9, 9E9]];
	VAR jointtarget CDP_3886 := [[2.86, 35.18, 6.96, 0, 47.86, -267.14], [9E9, 9E9, 9E9, 9E9, 9E9, 9E9]];
